LIN {X 0,Y 691.655,Z 288.187,A -85,B 0,C 180,E1 31271.101,E2 31271.101} C_VEL
LIN {X 0,Y 692.727,Z 290.872,A -85,B 0,C 180,E1 31270.983,E2 31270.983} C_VEL
LIN {X 0,Y 697.002,Z 308.209,A -85,B 0,C 180,E1 31270.448,E2 31270.448} C_VEL
LIN {X 0,Y 694.595,Z 554.038,A -85,B 0,C 180,E1 31267.412,E2 31267.412} C_VEL
LIN {X 0,Y 693.004,Z 720.794,A -85,B 0,C 180,E1 31265.381,E2 31265.381} C_VEL
LIN {X 0,Y 692.454,Z 746.763,A -85,B 0,C 180,E1 31264.93,E2 31264.93} C_VEL
LIN {X 0,Y 691.672,Z 770.938,A -85,B 0,C 180,E1 31264.354,E2 31264.354} C_VEL
LIN {X 0,Y 690.893,Z 792.668,A -85,B 0,C 180,E1 31263.712,E2 31263.712} C_VEL
LIN {X 0,Y 689.877,Z 818.249,A -85,B 0,C 180,E1 31262.792,E2 31262.792} C_VEL
LIN {X 0,Y 688.879,Z 840.235,A -85,B 0,C 180,E1 31261.844,E2 31261.844} C_VEL
LIN {X 0,Y 687.927,Z 859.99,A -85,B 0,C 180,E1 31260.869,E2 31260.869} C_VEL
LIN {X 0,Y 686.715,Z 883.646,A -85,B 0,C 180,E1 31259.529,E2 31259.529} C_VEL
LIN {X 0,Y 685.722,Z 903.008,A -85,B 0,C 180,E1 31258.269,E2 31258.269} C_VEL
LIN {X 0,Y 684.739,Z 922.512,A -85,B 0,C 180,E1 31256.847,E2 31256.847} C_VEL
LIN {X 0,Y 683.705,Z 942.533,A -85,B 0,C 180,E1 31255.187,E2 31255.187} C_VEL
LIN {X 0,Y 682.935,Z 959.025,A -85,B 0,C 180,E1 31253.651,E2 31253.651} C_VEL
LIN {X 0,Y 682.076,Z 977.766,A -85,B 0,C 180,E1 31251.68,E2 31251.68} C_VEL
LIN {X 0,Y 681.526,Z 991.915,A -85,B 0,C 180,E1 31249.989,E2 31249.989} C_VEL
LIN {X 0,Y 680.987,Z 1006.96,A -85,B 0,C 180,E1 31247.959,E2 31247.959} C_VEL
LIN {X 0,Y 680.597,Z 1019.263,A -85,B 0,C 180,E1 31246.033,E2 31246.033} C_VEL
LIN {X 0,Y 680.349,Z 1029.493,A -85,B 0,C 180,E1 31244.208,E2 31244.208} C_VEL
LIN {X 0,Y 680.126,Z 1040.171,A -85,B 0,C 180,E1 31241.964,E2 31241.964} C_VEL
LIN {X 0,Y 680.014,Z 1047.574,A -85,B 0,C 180,E1 31240.077,E2 31240.077} C_VEL
LIN {X 0,Y 679.956,Z 1053.149,A -85,B 0,C 180,E1 31238.371,E2 31238.371} C_VEL
LIN {X 0,Y 679.934,Z 1058.066,A -85,B 0,C 180,E1 31236.502,E2 31236.502} C_VEL
LIN {X 0,Y 679.908,Z 1062.337,A -85,B 0,C 180,E1 31234.217,E2 31234.217} C_VEL
LIN {X 0,Y 679.903,Z 1064.439,A -85,B 0,C 180,E1 31232.36,E2 31232.36} C_VEL
LIN {X 0,Y 679.893,Z 1065.35,A -85,B 0,C 180,E1 31230.59,E2 31230.59} C_VEL
LIN {X 0,Y 679.896,Z 1065.1,A -85,B 0,C 180,E1 31228.483,E2 31228.483} C_VEL
LIN {X 0,Y 679.907,Z 1063.128,A -85,B 0,C 180,E1 31226.374,E2 31226.374} C_VEL
LIN {X 0,Y 679.906,Z 1060.326,A -85,B 0,C 180,E1 31224.599,E2 31224.599} C_VEL
LIN {X 0,Y 679.946,Z 1056.414,A -85,B 0,C 180,E1 31222.82,E2 31222.82} C_VEL
LIN {X 0,Y 679.996,Z 1050.101,A -85,B 0,C 180,E1 31220.634,E2 31220.634} C_VEL
LIN {X 0,Y 680.095,Z 1042.663,A -85,B 0,C 180,E1 31218.638,E2 31218.638} C_VEL
LIN {X 0,Y 680.243,Z 1034.661,A -85,B 0,C 180,E1 31216.831,E2 31216.831} C_VEL
LIN {X 0,Y 680.475,Z 1023.917,A -85,B 0,C 180,E1 31214.751,E2 31214.751} C_VEL
LIN {X 0,Y 680.821,Z 1011.607,A -85,B 0,C 180,E1 31212.743,E2 31212.743} C_VEL
LIN {X 0,Y 681.259,Z 999.084,A -85,B 0,C 180,E1 31210.946,E2 31210.946} C_VEL
LIN {X 0,Y 681.869,Z 983.192,A -85,B 0,C 180,E1 31208.945,E2 31208.945} C_VEL
LIN {X 0,Y 682.513,Z 967.869,A -85,B 0,C 180,E1 31207.247,E2 31207.247} C_VEL
LIN {X 0,Y 683.4,Z 949.629,A -85,B 0,C 180,E1 31205.448,E2 31205.448} C_VEL
LIN {X 0,Y 684.27,Z 931.318,A -85,B 0,C 180,E1 31203.86,E2 31203.86} C_VEL
LIN {X 0,Y 685.293,Z 911.624,A -85,B 0,C 180,E1 31202.333,E2 31202.333} C_VEL
LIN {X 0,Y 686.389,Z 890.241,A -85,B 0,C 180,E1 31200.886,E2 31200.886} C_VEL
LIN {X 0,Y 687.364,Z 871.013,A -85,B 0,C 180,E1 31199.732,E2 31199.732} C_VEL
LIN {X 0,Y 688.556,Z 847.098,A -85,B 0,C 180,E1 31198.476,E2 31198.476} C_VEL
LIN {X 0,Y 689.557,Z 825.428,A -85,B 0,C 180,E1 31197.504,E2 31197.504} C_VEL
LIN {X 0,Y 690.438,Z 804.966,A -85,B 0,C 180,E1 31196.711,E2 31196.711} C_VEL
LIN {X 0,Y 691.403,Z 780.267,A -85,B 0,C 180,E1 31195.902,E2 31195.902} C_VEL
LIN {X 0,Y 692.129,Z 755.448,A -85,B 0,C 180,E1 31195.261,E2 31195.261} C_VEL
LIN {X 0,Y 692.718,Z 733.155,A -85,B 0,C 180,E1 31194.813,E2 31194.813} C_VEL
LIN {X 0,Y 693.254,Z 702.79,A -85,B 0,C 180,E1 31194.382,E2 31194.382} C_VEL
LIN {X 0,Y 695.461,Z 462.135,A -85,B 0,C 180,E1 31191.463,E2 31191.463} C_VEL
LIN {X 0,Y 696.866,Z 306.943,A -85,B 0,C 180,E1 31189.526,E2 31189.526} C_VEL
LIN {X 0,Y 691.957,Z 288.727,A -85,B 0,C 180,E1 31188.933,E2 31188.933} C_VEL
LIN {X 0,Y 690.695,Z 285.865,A -85,B 0,C 180,E1 31188.69,E2 31188.69} C_VEL
LIN {X 0,Y 681.985,Z 265.035,A -85,B 0,C 180,E1 31186.409,E2 31186.409} C_VEL
LIN {X 0,Y 680.481,Z 261.414,A -85,B 0,C 180,E1 31185.961,E2 31185.961} C_VEL
LIN {X 0,Y 680.519,Z 261.191,A -85,B 0,C 180,E1 31183.212,E2 31183.212} C_VEL
LIN {X 0,Y 680.458,Z 261.216,A -85,B 0,C 180,E1 31180.282,E2 31180.282} C_VEL
LIN {X 0,Y 680.458,Z 261.206,A -85,B 0,C 180,E1 31177.683,E2 31177.683} C_VEL
LIN {X 0,Y 680.502,Z 261.193,A -85,B 0,C 180,E1 31174.631,E2 31174.631} C_VEL
LIN {X 0,Y 680.449,Z 261.216,A -85,B 0,C 180,E1 31171.839,E2 31171.839} C_VEL
LIN {X 0,Y 680.517,Z 261.192,A -85,B 0,C 180,E1 31169.004,E2 31169.004} C_VEL
LIN {X 0,Y 680.459,Z 261.217,A -85,B 0,C 180,E1 31166.063,E2 31166.063} C_VEL
LIN {X 0,Y 680.458,Z 261.208,A -85,B 0,C 180,E1 31163.467,E2 31163.467} C_VEL
LIN {X 0,Y 680.512,Z 261.209,A -85,B 0,C 180,E1 31160.469,E2 31160.469} C_VEL
LIN {X 0,Y 680.45,Z 261.214,A -85,B 0,C 180,E1 31157.709,E2 31157.709} C_VEL
LIN {X 0,Y 680.488,Z 261.211,A -85,B 0,C 180,E1 31154.988,E2 31154.988} C_VEL
LIN {X 0,Y 680.467,Z 261.215,A -85,B 0,C 180,E1 31151.958,E2 31151.958} C_VEL
LIN {X 0,Y 680.454,Z 261.212,A -85,B 0,C 180,E1 31149.302,E2 31149.302} C_VEL
LIN {X 0,Y 680.524,Z 261.216,A -85,B 0,C 180,E1 31146.327,E2 31146.327} C_VEL
LIN {X 0,Y 680.449,Z 261.212,A -85,B 0,C 180,E1 31143.454,E2 31143.454} C_VEL
LIN {X 0,Y 680.498,Z 261.211,A -85,B 0,C 180,E1 31140.674,E2 31140.674} C_VEL
LIN {X 0,Y 680.46,Z 261.216,A -85,B 0,C 180,E1 31137.642,E2 31137.642} C_VEL
LIN {X 0,Y 680.455,Z 261.207,A -85,B 0,C 180,E1 31135.026,E2 31135.026} C_VEL
LIN {X 0,Y 680.514,Z 261.208,A -85,B 0,C 180,E1 31132.018,E2 31132.018} C_VEL
LIN {X 0,Y 680.449,Z 261.215,A -85,B 0,C 180,E1 31129.244,E2 31129.244} C_VEL
LIN {X 0,Y 680.48,Z 261.204,A -85,B 0,C 180,E1 31126.575,E2 31126.575} C_VEL
LIN {X 0,Y 680.468,Z 261.208,A -85,B 0,C 180,E1 31123.525,E2 31123.525} C_VEL
LIN {X 0,Y 680.451,Z 261.215,A -85,B 0,C 180,E1 31120.871,E2 31120.871} C_VEL
LIN {X 0,Y 680.53,Z 261.209,A -85,B 0,C 180,E1 31117.905,E2 31117.905} C_VEL
LIN {X 0,Y 680.447,Z 261.201,A -85,B 0,C 180,E1 31115.046,E2 31115.046} C_VEL
LIN {X 0,Y 680.479,Z 261.193,A -85,B 0,C 180,E1 31112.333,E2 31112.333} C_VEL
LIN {X 0,Y 680.498,Z 261.213,A -85,B 0,C 180,E1 31109.544,E2 31109.544} C_VEL
LIN {X 0,Y 679.438,Z 261.336,A -85,B 0,C 180,E1 31108.895,E2 31108.895} C_VEL
LIN {X 0,Y 673.022,Z 262.111,A -85,B 0,C 180,E1 31107.077,E2 31107.077} C_VEL
LIN {X 0,Y 672.51,Z 262.173,A -85,B 0,C 180,E1 31106.605,E2 31106.605} C_VEL
LIN {X 0,Y 672.581,Z 262.203,A -85,B 0,C 180,E1 31103.617,E2 31103.617} C_VEL
LIN {X 0,Y 672.511,Z 262.207,A -85,B 0,C 180,E1 31100.77,E2 31100.77} C_VEL
LIN {X 0,Y 672.551,Z 262.199,A -85,B 0,C 180,E1 31098.018,E2 31098.018} C_VEL
LIN {X 0,Y 672.519,Z 262.211,A -85,B 0,C 180,E1 31094.928,E2 31094.928} C_VEL
LIN {X 0,Y 672.516,Z 262.211,A -85,B 0,C 180,E1 31092.339,E2 31092.339} C_VEL
LIN {X 0,Y 672.546,Z 262.409,A -85,B 0,C 180,E1 31090.822,E2 31090.822} C_VEL
LIN {X 0,Y 675.389,Z 269.32,A -85,B 0,C 180,E1 31089.98,E2 31089.98} C_VEL
LIN {X 0,Y 679.147,Z 278.36,A -85,B 0,C 180,E1 31088.98,E2 31088.98} C_VEL
LIN {X 0,Y 689.647,Z 295.139,A -85,B 0,C 180,E1 31087.967,E2 31087.967} C_VEL
LIN {X 0,Y 690.879,Z 300.784,A -85,B 0,C 180,E1 31087.802,E2 31087.802} C_VEL
LIN {X 0,Y 688.209,Z 546.789,A -85,B 0,C 180,E1 31084.739,E2 31084.739} C_VEL
LIN {X 0,Y 686.469,Z 710.938,A -85,B 0,C 180,E1 31082.722,E2 31082.722} C_VEL
LIN {X 0,Y 685.844,Z 737.281,A -85,B 0,C 180,E1 31082.259,E2 31082.259} C_VEL
LIN {X 0,Y 685.014,Z 760.984,A -85,B 0,C 180,E1 31081.689,E2 31081.689} C_VEL
LIN {X 0,Y 684.18,Z 782.262,A -85,B 0,C 180,E1 31081.057,E2 31081.057} C_VEL
LIN {X 0,Y 683.101,Z 806.64,A -85,B 0,C 180,E1 31080.185,E2 31080.185} C_VEL
LIN {X 0,Y 681.937,Z 829.91,A -85,B 0,C 180,E1 31079.178,E2 31079.178} C_VEL
LIN {X 0,Y 680.867,Z 850.113,A -85,B 0,C 180,E1 31078.173,E2 31078.173} C_VEL
LIN {X 0,Y 679.511,Z 873.951,A -85,B 0,C 180,E1 31076.808,E2 31076.808} C_VEL
LIN {X 0,Y 678.374,Z 893.92,A -85,B 0,C 180,E1 31075.492,E2 31075.492} C_VEL
LIN {X 0,Y 677.213,Z 914.8,A -85,B 0,C 180,E1 31073.944,E2 31073.944} C_VEL
LIN {X 0,Y 676.092,Z 934.087,A -85,B 0,C 180,E1 31072.302,E2 31072.302} C_VEL
LIN {X 0,Y 675.237,Z 950.678,A -85,B 0,C 180,E1 31070.727,E2 31070.727} C_VEL
LIN {X 0,Y 674.302,Z 968.848,A -85,B 0,C 180,E1 31068.77,E2 31068.77} C_VEL
LIN {X 0,Y 673.674,Z 983.352,A -85,B 0,C 180,E1 31067.001,E2 31067.001} C_VEL
LIN {X 0,Y 673.066,Z 998.525,A -85,B 0,C 180,E1 31064.892,E2 31064.892} C_VEL
LIN {X 0,Y 672.666,Z 1009.999,A -85,B 0,C 180,E1 31063.058,E2 31063.058} C_VEL
LIN {X 0,Y 672.371,Z 1020.927,A -85,B 0,C 180,E1 31061.06,E2 31061.06} C_VEL
LIN {X 0,Y 672.144,Z 1030.836,A -85,B 0,C 180,E1 31058.9,E2 31058.9} C_VEL
LIN {X 0,Y 672.028,Z 1037.897,A -85,B 0,C 180,E1 31057.061,E2 31057.061} C_VEL
LIN {X 0,Y 671.964,Z 1043.795,A -85,B 0,C 180,E1 31055.208,E2 31055.208} C_VEL
LIN {X 0,Y 671.918,Z 1049.432,A -85,B 0,C 180,E1 31052.9,E2 31052.9} C_VEL
LIN {X 0,Y 671.919,Z 1052.713,A -85,B 0,C 180,E1 31050.938,E2 31050.938} C_VEL
LIN {X 0,Y 671.906,Z 1054.593,A -85,B 0,C 180,E1 31049.147,E2 31049.147} C_VEL
LIN {X 0,Y 671.908,Z 1055.491,A -85,B 0,C 180,E1 31047.014,E2 31047.014} C_VEL
LIN {X 0,Y 671.909,Z 1054.684,A -85,B 0,C 180,E1 31044.877,E2 31044.877} C_VEL
LIN {X 0,Y 671.917,Z 1052.852,A -85,B 0,C 180,E1 31043.077,E2 31043.077} C_VEL
LIN {X 0,Y 671.908,Z 1049.717,A -85,B 0,C 180,E1 31041.162,E2 31041.162} C_VEL
LIN {X 0,Y 671.96,Z 1044.22,A -85,B 0,C 180,E1 31038.846,E2 31038.846} C_VEL
LIN {X 0,Y 672.019,Z 1038.182,A -85,B 0,C 180,E1 31036.929,E2 31036.929} C_VEL
LIN {X 0,Y 672.14,Z 1031.512,A -85,B 0,C 180,E1 31035.175,E2 31035.175} C_VEL
LIN {X 0,Y 672.345,Z 1021.978,A -85,B 0,C 180,E1 31033.053,E2 31033.053} C_VEL
LIN {X 0,Y 672.658,Z 1010.349,A -85,B 0,C 180,E1 31030.912,E2 31030.912} C_VEL
LIN {X 0,Y 673.042,Z 999.136,A -85,B 0,C 180,E1 31029.112,E2 31029.112} C_VEL
LIN {X 0,Y 673.653,Z 983.784,A -85,B 0,C 180,E1 31026.964,E2 31026.964} C_VEL
LIN {X 0,Y 674.284,Z 969.258,A -85,B 0,C 180,E1 31025.187,E2 31025.187} C_VEL
LIN {X 0,Y 675.169,Z 952.248,A -85,B 0,C 180,E1 31023.338,E2 31023.338} C_VEL
LIN {X 0,Y 676.04,Z 935.141,A -85,B 0,C 180,E1 31021.704,E2 31021.704} C_VEL
LIN {X 0,Y 677.004,Z 917.895,A -85,B 0,C 180,E1 31020.221,E2 31020.221} C_VEL
LIN {X 0,Y 678.281,Z 895.722,A -85,B 0,C 180,E1 31018.544,E2 31018.544} C_VEL
LIN {X 0,Y 679.361,Z 876.399,A -85,B 0,C 180,E1 31017.256,E2 31017.256} C_VEL
LIN {X 0,Y 680.736,Z 852.619,A -85,B 0,C 180,E1 31015.869,E2 31015.869} C_VEL
LIN {X 0,Y 681.857,Z 831.556,A -85,B 0,C 180,E1 31014.809,E2 31014.809} C_VEL
LIN {X 0,Y 682.86,Z 811.527,A -85,B 0,C 180,E1 31013.928,E2 31013.928} C_VEL
LIN {X 0,Y 683.98,Z 787.389,A -85,B 0,C 180,E1 31013.019,E2 31013.019} C_VEL
LIN {X 0,Y 684.916,Z 763.254,A -85,B 0,C 180,E1 31012.282,E2 31012.282} C_VEL
LIN {X 0,Y 685.669,Z 741.656,A -85,B 0,C 180,E1 31011.748,E2 31011.748} C_VEL
LIN {X 0,Y 686.413,Z 715.552,A -85,B 0,C 180,E1 31011.254,E2 31011.254} C_VEL
LIN {X 0,Y 686.973,Z 669.627,A -85,B 0,C 180,E1 31010.667,E2 31010.667} C_VEL
LIN {X 0,Y 689.295,Z 440.854,A -85,B 0,C 180,E1 31007.861,E2 31007.861} C_VEL
LIN {X 0,Y 690.73,Z 299.325,A -85,B 0,C 180,E1 31006.077,E2 31006.077} C_VEL
LIN {X 0,Y 689.212,Z 294.353,A -85,B 0,C 180,E1 31005.901,E2 31005.901} C_VEL
LIN {X 0,Y 678.836,Z 277.664,A -85,B 0,C 180,E1 31004.874,E2 31004.874} C_VEL
LIN {X 0,Y 673.637,Z 265.405,A -85,B 0,C 180,E1 31003.462,E2 31003.462} C_VEL
LIN {X 0,Y 672.543,Z 262.387,A -85,B 0,C 180,E1 31003.08,E2 31003.08} C_VEL
LIN {X 0,Y 672.584,Z 262.19,A -85,B 0,C 180,E1 31000.17,E2 31000.17} C_VEL
LIN {X 0,Y 672.509,Z 262.194,A -85,B 0,C 180,E1 30997.303,E2 30997.303} C_VEL
LIN {X 0,Y 672.555,Z 262.193,A -85,B 0,C 180,E1 30994.55,E2 30994.55} C_VEL
LIN {X 0,Y 672.526,Z 262.2,A -85,B 0,C 180,E1 30991.557,E2 30991.557} C_VEL
LIN {X 0,Y 672.511,Z 262.204,A -85,B 0,C 180,E1 30988.993,E2 30988.993} C_VEL
LIN {X 0,Y 672.585,Z 262.176,A -85,B 0,C 180,E1 30986.107,E2 30986.107} C_VEL
LIN {X 0,Y 672.513,Z 262.204,A -85,B 0,C 180,E1 30983.204,E2 30983.204} C_VEL
LIN {X 0,Y 672.521,Z 262.188,A -85,B 0,C 180,E1 30980.632,E2 30980.632} C_VEL
LIN {X 0,Y 672.54,Z 262.203,A -85,B 0,C 180,E1 30977.477,E2 30977.477} C_VEL
LIN {X 0,Y 672.51,Z 262.195,A -85,B 0,C 180,E1 30974.817,E2 30974.817} C_VEL
LIN {X 0,Y 672.585,Z 262.19,A -85,B 0,C 180,E1 30971.926,E2 30971.926} C_VEL
LIN {X 0,Y 672.512,Z 262.198,A -85,B 0,C 180,E1 30968.981,E2 30968.981} C_VEL
LIN {X 0,Y 672.52,Z 262.174,A -85,B 0,C 180,E1 30966.402,E2 30966.402} C_VEL
LIN {X 0,Y 672.55,Z 262.2,A -85,B 0,C 180,E1 30963.324,E2 30963.324} C_VEL
LIN {X 0,Y 672.509,Z 262.185,A -85,B 0,C 180,E1 30960.596,E2 30960.596} C_VEL
LIN {X 0,Y 672.585,Z 262.196,A -85,B 0,C 180,E1 30957.7,E2 30957.7} C_VEL
LIN {X 0,Y 672.513,Z 262.195,A -85,B 0,C 180,E1 30954.711,E2 30954.711} C_VEL
LIN {X 0,Y 672.53,Z 262.178,A -85,B 0,C 180,E1 30952.052,E2 30952.052} C_VEL
LIN {X 0,Y 672.53,Z 262.199,A -85,B 0,C 180,E1 30948.889,E2 30948.889} C_VEL
LIN {X 0,Y 672.511,Z 262.177,A -85,B 0,C 180,E1 30946.238,E2 30946.238} C_VEL
LIN {X 0,Y 672.588,Z 262.201,A -85,B 0,C 180,E1 30943.326,E2 30943.326} C_VEL
LIN {X 0,Y 672.512,Z 262.186,A -85,B 0,C 180,E1 30940.456,E2 30940.456} C_VEL
LIN {X 0,Y 672.544,Z 262.196,A -85,B 0,C 180,E1 30937.721,E2 30937.721} C_VEL
LIN {X 0,Y 672.53,Z 262.199,A -85,B 0,C 180,E1 30934.647,E2 30934.647} C_VEL
LIN {X 0,Y 672.517,Z 262.203,A -85,B 0,C 180,E1 30931.977,E2 30931.977} C_VEL
LIN {X 0,Y 672.587,Z 262.19,A -85,B 0,C 180,E1 30929.044,E2 30929.044} C_VEL
LIN {X 0,Y 672.511,Z 262.191,A -85,B 0,C 180,E1 30926.113,E2 30926.113} C_VEL
LIN {X 0,Y 672.575,Z 262.186,A -85,B 0,C 180,E1 30923.255,E2 30923.255} C_VEL
LIN {X 0,Y 672.518,Z 262.206,A -85,B 0,C 180,E1 30920.234,E2 30920.234} C_VEL
LIN {X 0,Y 672.522,Z 262.208,A -85,B 0,C 180,E1 30917.64,E2 30917.64} C_VEL
LIN {X 0,Y 672.591,Z 262.407,A -85,B 0,C 180,E1 30914.594,E2 30914.594} C_VEL
LIN {X 0,Y 675.087,Z 268.808,A -85,B 0,C 180,E1 30913.837,E2 30913.837} C_VEL
LIN {X 0,Y 682.354,Z 285.802,A -85,B 0,C 180,E1 30911.928,E2 30911.928} C_VEL
LIN {X 0,Y 683.711,Z 288.641,A -85,B 0,C 180,E1 30911.673,E2 30911.673} C_VEL
LIN {X 0,Y 687.061,Z 294.502,A -85,B 0,C 180,E1 30911.345,E2 30911.345} C_VEL
LIN {X 0,Y 690.886,Z 310.252,A -85,B 0,C 180,E1 30910.854,E2 30910.854} C_VEL
LIN {X 0,Y 688.219,Z 556.025,A -85,B 0,C 180,E1 30907.794,E2 30907.794} C_VEL
LIN {X 0,Y 686.47,Z 720.881,A -85,B 0,C 180,E1 30905.768,E2 30905.768} C_VEL
LIN {X 0,Y 685.855,Z 747.02,A -85,B 0,C 180,E1 30905.31,E2 30905.31} C_VEL
LIN {X 0,Y 685.017,Z 770.919,A -85,B 0,C 180,E1 30904.735,E2 30904.735} C_VEL
LIN {X 0,Y 684.196,Z 791.933,A -85,B 0,C 180,E1 30904.112,E2 30904.112} C_VEL
LIN {X 0,Y 683.116,Z 816.377,A -85,B 0,C 180,E1 30903.241,E2 30903.241} C_VEL
LIN {X 0,Y 681.971,Z 839.227,A -85,B 0,C 180,E1 30902.255,E2 30902.255} C_VEL
LIN {X 0,Y 680.932,Z 858.899,A -85,B 0,C 180,E1 30901.282,E2 30901.282} C_VEL
LIN {X 0,Y 679.639,Z 882.174,A -85,B 0,C 180,E1 30899.965,E2 30899.965} C_VEL
LIN {X 0,Y 678.402,Z 903.283,A -85,B 0,C 180,E1 30898.582,E2 30898.582} C_VEL
LIN {X 0,Y 677.289,Z 923.369,A -85,B 0,C 180,E1 30897.099,E2 30897.099} C_VEL
LIN {X 0,Y 676.158,Z 942.892,A -85,B 0,C 180,E1 30895.455,E2 30895.455} C_VEL
LIN {X 0,Y 675.305,Z 959.023,A -85,B 0,C 180,E1 30893.935,E2 30893.935} C_VEL
LIN {X 0,Y 674.352,Z 977.768,A -85,B 0,C 180,E1 30891.941,E2 30891.941} C_VEL
LIN {X 0,Y 673.737,Z 991.914,A -85,B 0,C 180,E1 30890.23,E2 30890.23} C_VEL
LIN {X 0,Y 673.124,Z 1006.962,A -85,B 0,C 180,E1 30888.176,E2 30888.176} C_VEL
LIN {X 0,Y 672.684,Z 1019.35,A -85,B 0,C 180,E1 30886.213,E2 30886.213} C_VEL
LIN {X 0,Y 672.41,Z 1029.491,A -85,B 0,C 180,E1 30884.379,E2 30884.379} C_VEL
LIN {X 0,Y 672.157,Z 1040.172,A -85,B 0,C 180,E1 30882.108,E2 30882.108} C_VEL
LIN {X 0,Y 672.037,Z 1047.574,A -85,B 0,C 180,E1 30880.198,E2 30880.198} C_VEL
LIN {X 0,Y 671.961,Z 1053.405,A -85,B 0,C 180,E1 30878.385,E2 30878.385} C_VEL
LIN {X 0,Y 671.932,Z 1058.885,A -85,B 0,C 180,E1 30876.236,E2 30876.236} C_VEL
LIN {X 0,Y 671.913,Z 1062.564,A -85,B 0,C 180,E1 30874.096,E2 30874.096} C_VEL
LIN {X 0,Y 671.904,Z 1064.506,A -85,B 0,C 180,E1 30872.303,E2 30872.303} C_VEL
LIN {X 0,Y 671.892,Z 1065.395,A -85,B 0,C 180,E1 30870.426,E2 30870.426} C_VEL
LIN {X 0,Y 671.904,Z 1064.842,A -85,B 0,C 180,E1 30868.124,E2 30868.124} C_VEL
LIN {X 0,Y 671.911,Z 1063.015,A -85,B 0,C 180,E1 30866.246,E2 30866.246} C_VEL
LIN {X 0,Y 671.903,Z 1060.167,A -85,B 0,C 180,E1 30864.449,E2 30864.449} C_VEL
LIN {X 0,Y 671.949,Z 1056,A -85,B 0,C 180,E1 30862.562,E2 30862.562} C_VEL
LIN {X 0,Y 671.999,Z 1049.094,A -85,B 0,C 180,E1 30860.234,E2 30860.234} C_VEL
LIN {X 0,Y 672.131,Z 1042.308,A -85,B 0,C 180,E1 30858.415,E2 30858.415} C_VEL
LIN {X 0,Y 672.3,Z 1034.214,A -85,B 0,C 180,E1 30856.576,E2 30856.576} C_VEL
LIN {X 0,Y 672.597,Z 1022.886,A -85,B 0,C 180,E1 30854.391,E2 30854.391} C_VEL
LIN {X 0,Y 672.965,Z 1011.028,A -85,B 0,C 180,E1 30852.445,E2 30852.445} C_VEL
LIN {X 0,Y 673.481,Z 997.688,A -85,B 0,C 180,E1 30850.521,E2 30850.521} C_VEL
LIN {X 0,Y 674.192,Z 981.649,A -85,B 0,C 180,E1 30848.511,E2 30848.511} C_VEL
LIN {X 0,Y 674.879,Z 967.018,A -85,B 0,C 180,E1 30846.883,E2 30846.883} C_VEL
LIN {X 0,Y 675.928,Z 947.6,A -85,B 0,C 180,E1 30844.971,E2 30844.971} C_VEL
LIN {X 0,Y 676.829,Z 930.762,A -85,B 0,C 180,E1 30843.503,E2 30843.503} C_VEL
LIN {X 0,Y 678.02,Z 910.69,A -85,B 0,C 180,E1 30841.938,E2 30841.938} C_VEL
LIN {X 0,Y 679.23,Z 888.897,A -85,B 0,C 180,E1 30840.46,E2 30840.46} C_VEL
LIN {X 0,Y 680.369,Z 868.576,A -85,B 0,C 180,E1 30839.241,E2 30839.241} C_VEL
LIN {X 0,Y 681.735,Z 843.973,A -85,B 0,C 180,E1 30837.968,E2 30837.968} C_VEL
LIN {X 0,Y 682.775,Z 823.343,A -85,B 0,C 180,E1 30837.049,E2 30837.049} C_VEL
LIN {X 0,Y 683.767,Z 802.394,A -85,B 0,C 180,E1 30836.242,E2 30836.242} C_VEL
LIN {X 0,Y 684.827,Z 775.425,A -85,B 0,C 180,E1 30835.386,E2 30835.386} C_VEL
LIN {X 0,Y 685.596,Z 753.439,A -85,B 0,C 180,E1 30834.832,E2 30834.832} C_VEL
LIN {X 0,Y 686.302,Z 729.652,A -85,B 0,C 180,E1 30834.365,E2 30834.365} C_VEL
LIN {X 0,Y 686.824,Z 694.807,A -85,B 0,C 180,E1 30833.896,E2 30833.896} C_VEL
LIN {X 0,Y 689.235,Z 458.322,A -85,B 0,C 180,E1 30831,E2 30831} C_VEL
LIN {X 0,Y 690.749,Z 308.953,A -85,B 0,C 180,E1 30829.119,E2 30829.119} C_VEL
LIN {X 0,Y 686.523,Z 293.151,A -85,B 0,C 180,E1 30828.597,E2 30828.597} C_VEL
LIN {X 0,Y 683.09,Z 287.391,A -85,B 0,C 180,E1 30828.24,E2 30828.24} C_VEL
LIN {X 0,Y 675.482,Z 269.508,A -85,B 0,C 180,E1 30826.251,E2 30826.251} C_VEL
LIN {X 0,Y 672.607,Z 262.52,A -85,B 0,C 180,E1 30825.425,E2 30825.425} C_VEL
LIN {X 0,Y 672.54,Z 262.207,A -85,B 0,C 180,E1 30824.591,E2 30824.591} C_VEL
LIN {X 0,Y 672.515,Z 262.193,A -85,B 0,C 180,E1 30821.851,E2 30821.851} C_VEL
LIN {X 0,Y 672.584,Z 262.177,A -85,B 0,C 180,E1 30818.856,E2 30818.856} C_VEL
LIN {X 0,Y 672.513,Z 262.205,A -85,B 0,C 180,E1 30815.965,E2 30815.965} C_VEL
LIN {X 0,Y 672.564,Z 262.18,A -85,B 0,C 180,E1 30813.168,E2 30813.168} C_VEL
LIN {X 0,Y 672.521,Z 262.196,A -85,B 0,C 180,E1 30810.168,E2 30810.168} C_VEL
LIN {X 0,Y 672.518,Z 262.19,A -85,B 0,C 180,E1 30807.542,E2 30807.542} C_VEL
LIN {X 0,Y 672.57,Z 262.198,A -85,B 0,C 180,E1 30804.506,E2 30804.506} C_VEL
LIN {X 0,Y 672.512,Z 262.204,A -85,B 0,C 180,E1 30801.729,E2 30801.729} C_VEL
LIN {X 0,Y 672.568,Z 262.198,A -85,B 0,C 180,E1 30798.911,E2 30798.911} C_VEL
LIN {X 0,Y 672.517,Z 262.203,A -85,B 0,C 180,E1 30795.857,E2 30795.857} C_VEL
LIN {X 0,Y 672.522,Z 262.2,A -85,B 0,C 180,E1 30793.236,E2 30793.236} C_VEL
LIN {X 0,Y 672.547,Z 262.204,A -85,B 0,C 180,E1 30790.104,E2 30790.104} C_VEL
LIN {X 0,Y 672.51,Z 262.201,A -85,B 0,C 180,E1 30787.391,E2 30787.391} C_VEL
LIN {X 0,Y 672.585,Z 262.196,A -85,B 0,C 180,E1 30784.519,E2 30784.519} C_VEL
LIN {X 0,Y 672.513,Z 262.203,A -85,B 0,C 180,E1 30781.534,E2 30781.534} C_VEL
LIN {X 0,Y 672.529,Z 262.197,A -85,B 0,C 180,E1 30778.893,E2 30778.893} C_VEL
LIN {X 0,Y 672.531,Z 262.197,A -85,B 0,C 180,E1 30775.737,E2 30775.737} C_VEL
LIN {X 0,Y 672.512,Z 262.203,A -85,B 0,C 180,E1 30773.083,E2 30773.083} C_VEL
LIN {X 0,Y 672.588,Z 262.196,A -85,B 0,C 180,E1 30770.156,E2 30770.156} C_VEL
LIN {X 0,Y 672.51,Z 262.195,A -85,B 0,C 180,E1 30767.248,E2 30767.248} C_VEL
LIN {X 0,Y 672.53,Z 262.203,A -85,B 0,C 180,E1 30764.654,E2 30764.654} C_VEL
LIN {X 0,Y 672.527,Z 262.206,A -85,B 0,C 180,E1 30761.448,E2 30761.448} C_VEL
LIN {X 0,Y 672.515,Z 262.196,A -85,B 0,C 180,E1 30758.782,E2 30758.782} C_VEL
LIN {X 0,Y 672.577,Z 262.191,A -85,B 0,C 180,E1 30755.775,E2 30755.775} C_VEL
LIN {X 0,Y 672.507,Z 262.179,A -85,B 0,C 180,E1 30752.937,E2 30752.937} C_VEL
LIN {X 0,Y 672.552,Z 262.202,A -85,B 0,C 180,E1 30750.227,E2 30750.227} C_VEL
LIN {X 0,Y 672.516,Z 262.172,A -85,B 0,C 180,E1 30747.134,E2 30747.134} C_VEL
LIN {X 0,Y 672.51,Z 262.173,A -85,B 0,C 180,E1 30746.605,E2 30746.605} C_VEL
LIN {X 0,Y 671.56,Z 262.302,A -85,B 0,C 180,E1 30745.949,E2 30745.949} C_VEL
LIN {X 0,Y 665.112,Z 263.141,A -85,B 0,C 180,E1 30744.062,E2 30744.062} C_VEL
LIN {X 0,Y 664.643,Z 263.192,A -85,B 0,C 180,E1 30743.631,E2 30743.631} C_VEL
LIN {X 0,Y 664.572,Z 263.197,A -85,B 0,C 180,E1 30740.791,E2 30740.791} C_VEL
LIN {X 0,Y 664.605,Z 263.188,A -85,B 0,C 180,E1 30738.087,E2 30738.087} C_VEL
LIN {X 0,Y 664.586,Z 263.198,A -85,B 0,C 180,E1 30734.998,E2 30734.998} C_VEL
LIN {X 0,Y 664.575,Z 263.198,A -85,B 0,C 180,E1 30732.376,E2 30732.376} C_VEL
LIN {X 0,Y 664.685,Z 263.495,A -85,B 0,C 180,E1 30731.379,E2 30731.379} C_VEL
LIN {X 0,Y 670.815,Z 278.048,A -85,B 0,C 180,E1 30729.639,E2 30729.639} C_VEL
LIN {X 0,Y 684.181,Z 299.516,A -85,B 0,C 180,E1 30728.306,E2 30728.306} C_VEL
LIN {X 0,Y 684.794,Z 302.98,A -85,B 0,C 180,E1 30728.214,E2 30728.214} C_VEL
LIN {X 0,Y 681.873,Z 547.686,A -85,B 0,C 180,E1 30725.142,E2 30725.142} C_VEL
LIN {X 0,Y 679.968,Z 710.97,A -85,B 0,C 180,E1 30723.117,E2 30723.117} C_VEL
LIN {X 0,Y 679.28,Z 737.454,A -85,B 0,C 180,E1 30722.648,E2 30722.648} C_VEL
LIN {X 0,Y 678.393,Z 760.902,A -85,B 0,C 180,E1 30722.08,E2 30722.08} C_VEL
LIN {X 0,Y 677.559,Z 780.618,A -85,B 0,C 180,E1 30721.494,E2 30721.494} C_VEL
LIN {X 0,Y 676.486,Z 802.868,A -85,B 0,C 180,E1 30720.708,E2 30720.708} C_VEL
LIN {X 0,Y 675.119,Z 827.822,A -85,B 0,C 180,E1 30719.648,E2 30719.648} C_VEL
LIN {X 0,Y 673.935,Z 848.259,A -85,B 0,C 180,E1 30718.634,E2 30718.634} C_VEL
LIN {X 0,Y 672.584,Z 870.981,A -85,B 0,C 180,E1 30717.346,E2 30717.346} C_VEL
LIN {X 0,Y 671.148,Z 892.788,A -85,B 0,C 180,E1 30715.911,E2 30715.911} C_VEL
LIN {X 0,Y 669.994,Z 911.636,A -85,B 0,C 180,E1 30714.512,E2 30714.512} C_VEL
LIN {X 0,Y 668.709,Z 932.139,A -85,B 0,C 180,E1 30712.785,E2 30712.785} C_VEL
LIN {X 0,Y 667.726,Z 948.355,A -85,B 0,C 180,E1 30711.247,E2 30711.247} C_VEL
LIN {X 0,Y 666.762,Z 966.128,A -85,B 0,C 180,E1 30709.355,E2 30709.355} C_VEL
LIN {X 0,Y 665.988,Z 980.893,A -85,B 0,C 180,E1 30707.564,E2 30707.564} C_VEL
LIN {X 0,Y 665.367,Z 994.618,A -85,B 0,C 180,E1 30705.694,E2 30705.694} C_VEL
LIN {X 0,Y 664.827,Z 1008.169,A -85,B 0,C 180,E1 30703.569,E2 30703.569} C_VEL
LIN {X 0,Y 664.5,Z 1018.402,A -85,B 0,C 180,E1 30701.72,E2 30701.72} C_VEL
LIN {X 0,Y 664.231,Z 1028.467,A -85,B 0,C 180,E1 30699.619,E2 30699.619} C_VEL
LIN {X 0,Y 664.072,Z 1037.007,A -85,B 0,C 180,E1 30697.44,E2 30697.44} C_VEL
LIN {X 0,Y 663.966,Z 1042.891,A -85,B 0,C 180,E1 30695.617,E2 30695.617} C_VEL
LIN {X 0,Y 663.937,Z 1047.626,A -85,B 0,C 180,E1 30693.799,E2 30693.799} C_VEL
LIN {X 0,Y 663.897,Z 1051.969,A -85,B 0,C 180,E1 30691.553,E2 30691.553} C_VEL
LIN {X 0,Y 663.91,Z 1054.353,A -85,B 0,C 180,E1 30689.482,E2 30689.482} C_VEL
LIN {X 0,Y 663.896,Z 1055.322,A -85,B 0,C 180,E1 30687.669,E2 30687.669} C_VEL
LIN {X 0,Y 663.911,Z 1055.176,A -85,B 0,C 180,E1 30685.681,E2 30685.681} C_VEL
LIN {X 0,Y 663.907,Z 1053.371,A -85,B 0,C 180,E1 30683.427,E2 30683.427} C_VEL
LIN {X 0,Y 663.906,Z 1050.489,A -85,B 0,C 180,E1 30681.512,E2 30681.512} C_VEL
LIN {X 0,Y 663.949,Z 1046.802,A -85,B 0,C 180,E1 30679.764,E2 30679.764} C_VEL
LIN {X 0,Y 664.003,Z 1041.538,A -85,B 0,C 180,E1 30677.83,E2 30677.83} C_VEL
LIN {X 0,Y 664.139,Z 1033.33,A -85,B 0,C 180,E1 30675.482,E2 30675.482} C_VEL
LIN {X 0,Y 664.326,Z 1025.119,A -85,B 0,C 180,E1 30673.563,E2 30673.563} C_VEL
LIN {X 0,Y 664.586,Z 1015.231,A -85,B 0,C 180,E1 30671.582,E2 30671.582} C_VEL
LIN {X 0,Y 665.042,Z 1002.409,A -85,B 0,C 180,E1 30669.402,E2 30669.402} C_VEL
LIN {X 0,Y 665.563,Z 990.035,A -85,B 0,C 180,E1 30667.568,E2 30667.568} C_VEL
LIN {X 0,Y 666.337,Z 974.429,A -85,B 0,C 180,E1 30665.534,E2 30665.534} C_VEL
LIN {X 0,Y 667.122,Z 958.896,A -85,B 0,C 180,E1 30663.759,E2 30663.759} C_VEL
LIN {X 0,Y 668.19,Z 941.387,A -85,B 0,C 180,E1 30661.974,E2 30661.974} C_VEL
LIN {X 0,Y 669.303,Z 922.252,A -85,B 0,C 180,E1 30660.266,E2 30660.266} C_VEL
LIN {X 0,Y 670.438,Z 904.309,A -85,B 0,C 180,E1 30658.834,E2 30658.834} C_VEL
LIN {X 0,Y 671.894,Z 881.383,A -85,B 0,C 180,E1 30657.227,E2 30657.227} C_VEL
LIN {X 0,Y 673.073,Z 862.13,A -85,B 0,C 180,E1 30656.043,E2 30656.043} C_VEL
LIN {X 0,Y 674.532,Z 838.86,A -85,B 0,C 180,E1 30654.786,E2 30654.786} C_VEL
LIN {X 0,Y 675.825,Z 815.43,A -85,B 0,C 180,E1 30653.715,E2 30653.715} C_VEL
LIN {X 0,Y 676.85,Z 795.649,A -85,B 0,C 180,E1 30652.935,E2 30652.935} C_VEL
LIN {X 0,Y 677.876,Z 773.92,A -85,B 0,C 180,E1 30652.202,E2 30652.202} C_VEL
LIN {X 0,Y 678.875,Z 747.328,A -85,B 0,C 180,E1 30651.483,E2 30651.483} C_VEL
LIN {X 0,Y 679.574,Z 725.191,A -85,B 0,C 180,E1 30651.024,E2 30651.024} C_VEL
LIN {X 0,Y 680.197,Z 699.655,A -85,B 0,C 180,E1 30650.635,E2 30650.635} C_VEL
LIN {X 0,Y 682.922,Z 456.79,A -85,B 0,C 180,E1 30647.638,E2 30647.638} C_VEL
LIN {X 0,Y 684.655,Z 301.352,A -85,B 0,C 180,E1 30645.664,E2 30645.664} C_VEL
LIN {X 0,Y 683.59,Z 298.46,A -85,B 0,C 180,E1 30645.545,E2 30645.545} C_VEL
LIN {X 0,Y 670.7,Z 277.764,A -85,B 0,C 180,E1 30644.243,E2 30644.243} C_VEL
LIN {X 0,Y 664.682,Z 263.5,A -85,B 0,C 180,E1 30642.53,E2 30642.53} C_VEL
LIN {X 0,Y 664.571,Z 263.19,A -85,B 0,C 180,E1 30641.339,E2 30641.339} C_VEL
LIN {X 0,Y 664.63,Z 263.185,A -85,B 0,C 180,E1 30638.524,E2 30638.524} C_VEL
LIN {X 0,Y 664.58,Z 263.195,A -85,B 0,C 180,E1 30635.504,E2 30635.504} C_VEL
LIN {X 0,Y 664.579,Z 263.192,A -85,B 0,C 180,E1 30632.898,E2 30632.898} C_VEL
LIN {X 0,Y 664.625,Z 263.182,A -85,B 0,C 180,E1 30629.866,E2 30629.866} C_VEL
LIN {X 0,Y 664.572,Z 263.189,A -85,B 0,C 180,E1 30627.122,E2 30627.122} C_VEL
LIN {X 0,Y 664.635,Z 263.178,A -85,B 0,C 180,E1 30624.249,E2 30624.249} C_VEL
LIN {X 0,Y 664.578,Z 263.182,A -85,B 0,C 180,E1 30621.26,E2 30621.26} C_VEL
LIN {X 0,Y 664.585,Z 263.179,A -85,B 0,C 180,E1 30618.585,E2 30618.585} C_VEL
LIN {X 0,Y 664.601,Z 263.181,A -85,B 0,C 180,E1 30615.444,E2 30615.444} C_VEL
LIN {X 0,Y 664.57,Z 263.172,A -85,B 0,C 180,E1 30612.778,E2 30612.778} C_VEL
LIN {X 0,Y 664.65,Z 263.187,A -85,B 0,C 180,E1 30609.814,E2 30609.814} C_VEL
LIN {X 0,Y 664.569,Z 263.158,A -85,B 0,C 180,E1 30606.913,E2 30606.913} C_VEL
LIN {X 0,Y 664.597,Z 263.189,A -85,B 0,C 180,E1 30604.228,E2 30604.228} C_VEL
LIN {X 0,Y 664.584,Z 263.17,A -85,B 0,C 180,E1 30601.035,E2 30601.035} C_VEL
LIN {X 0,Y 664.578,Z 263.179,A -85,B 0,C 180,E1 30598.362,E2 30598.362} C_VEL
LIN {X 0,Y 664.631,Z 263.182,A -85,B 0,C 180,E1 30595.34,E2 30595.34} C_VEL
LIN {X 0,Y 664.568,Z 263.163,A -85,B 0,C 180,E1 30592.527,E2 30592.527} C_VEL
LIN {X 0,Y 664.636,Z 263.192,A -85,B 0,C 180,E1 30589.687,E2 30589.687} C_VEL
LIN {X 0,Y 664.577,Z 263.164,A -85,B 0,C 180,E1 30586.691,E2 30586.691} C_VEL
LIN {X 0,Y 664.587,Z 263.185,A -85,B 0,C 180,E1 30584.018,E2 30584.018} C_VEL
LIN {X 0,Y 664.599,Z 263.172,A -85,B 0,C 180,E1 30580.854,E2 30580.854} C_VEL
LIN {X 0,Y 664.574,Z 263.183,A -85,B 0,C 180,E1 30578.172,E2 30578.172} C_VEL
LIN {X 0,Y 664.651,Z 263.183,A -85,B 0,C 180,E1 30575.278,E2 30575.278} C_VEL
LIN {X 0,Y 664.575,Z 263.191,A -85,B 0,C 180,E1 30572.296,E2 30572.296} C_VEL
LIN {X 0,Y 664.604,Z 263.197,A -85,B 0,C 180,E1 30569.635,E2 30569.635} C_VEL
LIN {X 0,Y 664.584,Z 263.168,A -85,B 0,C 180,E1 30566.461,E2 30566.461} C_VEL
LIN {X 0,Y 664.579,Z 263.197,A -85,B 0,C 180,E1 30563.858,E2 30563.858} C_VEL
LIN {X 0,Y 664.636,Z 263.167,A -85,B 0,C 180,E1 30560.813,E2 30560.813} C_VEL
LIN {X 0,Y 664.574,Z 263.195,A -85,B 0,C 180,E1 30557.969,E2 30557.969} C_VEL
LIN {X 0,Y 664.663,Z 263.431,A -85,B 0,C 180,E1 30555.176,E2 30555.176} C_VEL
LIN {X 0,Y 673.862,Z 285.312,A -85,B 0,C 180,E1 30552.61,E2 30552.61} C_VEL
LIN {X 0,Y 675.209,Z 288.274,A -85,B 0,C 180,E1 30552.326,E2 30552.326} C_VEL
LIN {X 0,Y 681.574,Z 298.738,A -85,B 0,C 180,E1 30551.693,E2 30551.693} C_VEL
LIN {X 0,Y 684.804,Z 312.286,A -85,B 0,C 180,E1 30551.268,E2 30551.268} C_VEL
LIN {X 0,Y 681.881,Z 557.078,A -85,B 0,C 180,E1 30548.194,E2 30548.194} C_VEL
LIN {X 0,Y 679.969,Z 720.814,A -85,B 0,C 180,E1 30546.164,E2 30546.164} C_VEL
LIN {X 0,Y 679.293,Z 747.148,A -85,B 0,C 180,E1 30545.7,E2 30545.7} C_VEL
LIN {X 0,Y 678.402,Z 770.714,A -85,B 0,C 180,E1 30545.13,E2 30545.13} C_VEL
LIN {X 0,Y 677.532,Z 791.19,A -85,B 0,C 180,E1 30544.52,E2 30544.52} C_VEL
LIN {X 0,Y 676.433,Z 813.913,A -85,B 0,C 180,E1 30543.714,E2 30543.714} C_VEL
LIN {X 0,Y 675.098,Z 838.218,A -85,B 0,C 180,E1 30542.674,E2 30542.674} C_VEL
LIN {X 0,Y 673.94,Z 858.203,A -85,B 0,C 180,E1 30541.682,E2 30541.682} C_VEL
LIN {X 0,Y 672.605,Z 880.68,A -85,B 0,C 180,E1 30540.41,E2 30540.41} C_VEL
LIN {X 0,Y 671.209,Z 901.874,A -85,B 0,C 180,E1 30539.02,E2 30539.02} C_VEL
LIN {X 0,Y 670.057,Z 920.421,A -85,B 0,C 180,E1 30537.651,E2 30537.651} C_VEL
LIN {X 0,Y 668.75,Z 941.518,A -85,B 0,C 180,E1 30535.886,E2 30535.886} C_VEL
LIN {X 0,Y 667.738,Z 958.096,A -85,B 0,C 180,E1 30534.317,E2 30534.317} C_VEL
LIN {X 0,Y 666.809,Z 975.435,A -85,B 0,C 180,E1 30532.481,E2 30532.481} C_VEL
LIN {X 0,Y 665.974,Z 991.21,A -85,B 0,C 180,E1 30530.568,E2 30530.568} C_VEL
LIN {X 0,Y 665.346,Z 1005.108,A -85,B 0,C 180,E1 30528.669,E2 30528.669} C_VEL
LIN {X 0,Y 664.803,Z 1018.745,A -85,B 0,C 180,E1 30526.515,E2 30526.515} C_VEL
LIN {X 0,Y 664.485,Z 1029.031,A -85,B 0,C 180,E1 30524.643,E2 30524.643} C_VEL
LIN {X 0,Y 664.214,Z 1039.46,A -85,B 0,C 180,E1 30522.431,E2 30522.431} C_VEL
LIN {X 0,Y 664.067,Z 1047.27,A -85,B 0,C 180,E1 30520.41,E2 30520.41} C_VEL
LIN {X 0,Y 663.964,Z 1053.15,A -85,B 0,C 180,E1 30518.574,E2 30518.574} C_VEL
LIN {X 0,Y 663.936,Z 1058.066,A -85,B 0,C 180,E1 30516.659,E2 30516.659} C_VEL
LIN {X 0,Y 663.904,Z 1062.337,A -85,B 0,C 180,E1 30514.319,E2 30514.319} C_VEL
LIN {X 0,Y 663.905,Z 1064.439,A -85,B 0,C 180,E1 30512.417,E2 30512.417} C_VEL
LIN {X 0,Y 663.894,Z 1065.35,A -85,B 0,C 180,E1 30510.604,E2 30510.604} C_VEL
LIN {X 0,Y 663.895,Z 1065.099,A -85,B 0,C 180,E1 30508.447,E2 30508.447} C_VEL
LIN {X 0,Y 663.91,Z 1063.128,A -85,B 0,C 180,E1 30506.287,E2 30506.287} C_VEL
LIN {X 0,Y 663.905,Z 1060.326,A -85,B 0,C 180,E1 30504.469,E2 30504.469} C_VEL
LIN {X 0,Y 663.951,Z 1056.414,A -85,B 0,C 180,E1 30502.646,E2 30502.646} C_VEL
LIN {X 0,Y 664.009,Z 1050.306,A -85,B 0,C 180,E1 30500.466,E2 30500.466} C_VEL
LIN {X 0,Y 664.152,Z 1042.663,A -85,B 0,C 180,E1 30498.361,E2 30498.361} C_VEL
LIN {X 0,Y 664.337,Z 1034.537,A -85,B 0,C 180,E1 30496.482,E2 30496.482} C_VEL
LIN {X 0,Y 664.668,Z 1023.4,A -85,B 0,C 180,E1 30494.289,E2 30494.289} C_VEL
LIN {X 0,Y 665.075,Z 1011.607,A -85,B 0,C 180,E1 30492.321,E2 30492.321} C_VEL
LIN {X 0,Y 665.591,Z 999.366,A -85,B 0,C 180,E1 30490.519,E2 30490.519} C_VEL
LIN {X 0,Y 666.389,Z 983.188,A -85,B 0,C 180,E1 30488.432,E2 30488.432} C_VEL
LIN {X 0,Y 667.158,Z 968.308,A -85,B 0,C 180,E1 30486.741,E2 30486.741} C_VEL
LIN {X 0,Y 668.262,Z 950.135,A -85,B 0,C 180,E1 30484.901,E2 30484.901} C_VEL
LIN {X 0,Y 669.323,Z 931.87,A -85,B 0,C 180,E1 30483.278,E2 30483.278} C_VEL
LIN {X 0,Y 670.525,Z 913.13,A -85,B 0,C 180,E1 30481.79,E2 30481.79} C_VEL
LIN {X 0,Y 671.916,Z 890.973,A -85,B 0,C 180,E1 30480.246,E2 30480.246} C_VEL
LIN {X 0,Y 673.142,Z 870.925,A -85,B 0,C 180,E1 30479.018,E2 30479.018} C_VEL
LIN {X 0,Y 674.619,Z 847.224,A -85,B 0,C 180,E1 30477.753,E2 30477.753} C_VEL
LIN {X 0,Y 675.823,Z 825.421,A -85,B 0,C 180,E1 30476.759,E2 30476.759} C_VEL
LIN {X 0,Y 676.866,Z 805.349,A -85,B 0,C 180,E1 30475.969,E2 30475.969} C_VEL
LIN {X 0,Y 677.951,Z 782.316,A -85,B 0,C 180,E1 30475.196,E2 30475.196} C_VEL
LIN {X 0,Y 678.902,Z 756.539,A -85,B 0,C 180,E1 30474.51,E2 30474.51} C_VEL
LIN {X 0,Y 679.601,Z 734.474,A -85,B 0,C 180,E1 30474.056,E2 30474.056} C_VEL
LIN {X 0,Y 680.219,Z 707.836,A -85,B 0,C 180,E1 30473.657,E2 30473.657} C_VEL
LIN {X 0,Y 682.934,Z 465.741,A -85,B 0,C 180,E1 30470.669,E2 30470.669} C_VEL
LIN {X 0,Y 684.667,Z 310.936,A -85,B 0,C 180,E1 30468.704,E2 30468.704} C_VEL
LIN {X 0,Y 681.103,Z 297.645,A -85,B 0,C 180,E1 30468.257,E2 30468.257} C_VEL
LIN {X 0,Y 674.675,Z 287.31,A -85,B 0,C 180,E1 30467.599,E2 30467.599} C_VEL
LIN {X 0,Y 667.68,Z 270.691,A -85,B 0,C 180,E1 30465.712,E2 30465.712} C_VEL
LIN {X 0,Y 664.653,Z 263.381,A -85,B 0,C 180,E1 30464.808,E2 30464.808} C_VEL
LIN {X 0,Y 664.571,Z 263.176,A -85,B 0,C 180,E1 30462.031,E2 30462.031} C_VEL
LIN {X 0,Y 664.635,Z 263.168,A -85,B 0,C 180,E1 30459.187,E2 30459.187} C_VEL
LIN {X 0,Y 664.583,Z 263.196,A -85,B 0,C 180,E1 30456.248,E2 30456.248} C_VEL
LIN {X 0,Y 664.579,Z 263.169,A -85,B 0,C 180,E1 30453.62,E2 30453.62} C_VEL
LIN {X 0,Y 664.626,Z 263.186,A -85,B 0,C 180,E1 30450.564,E2 30450.564} C_VEL
LIN {X 0,Y 664.572,Z 263.179,A -85,B 0,C 180,E1 30447.788,E2 30447.788} C_VEL
LIN {X 0,Y 664.646,Z 263.192,A -85,B 0,C 180,E1 30444.886,E2 30444.886} C_VEL
LIN {X 0,Y 664.577,Z 263.194,A -85,B 0,C 180,E1 30441.909,E2 30441.909} C_VEL
LIN {X 0,Y 664.59,Z 263.188,A -85,B 0,C 180,E1 30439.238,E2 30439.238} C_VEL
LIN {X 0,Y 664.595,Z 263.191,A -85,B 0,C 180,E1 30436.071,E2 30436.071} C_VEL
LIN {X 0,Y 664.575,Z 263.19,A -85,B 0,C 180,E1 30433.397,E2 30433.397} C_VEL
LIN {X 0,Y 664.644,Z 263.194,A -85,B 0,C 180,E1 30430.401,E2 30430.401} C_VEL
LIN {X 0,Y 664.571,Z 263.191,A -85,B 0,C 180,E1 30427.521,E2 30427.521} C_VEL
LIN {X 0,Y 664.621,Z 263.188,A -85,B 0,C 180,E1 30424.746,E2 30424.746} C_VEL
LIN {X 0,Y 664.584,Z 263.193,A -85,B 0,C 180,E1 30421.724,E2 30421.724} C_VEL
LIN {X 0,Y 664.576,Z 263.187,A -85,B 0,C 180,E1 30419.138,E2 30419.138} C_VEL
LIN {X 0,Y 664.638,Z 263.184,A -85,B 0,C 180,E1 30416.118,E2 30416.118} C_VEL
LIN {X 0,Y 664.57,Z 263.193,A -85,B 0,C 180,E1 30413.26,E2 30413.26} C_VEL
LIN {X 0,Y 664.624,Z 263.181,A -85,B 0,C 180,E1 30410.474,E2 30410.474} C_VEL
LIN {X 0,Y 664.577,Z 263.184,A -85,B 0,C 180,E1 30407.399,E2 30407.399} C_VEL
LIN {X 0,Y 664.579,Z 263.193,A -85,B 0,C 180,E1 30404.824,E2 30404.824} C_VEL
LIN {X 0,Y 664.623,Z 263.193,A -85,B 0,C 180,E1 30401.764,E2 30401.764} C_VEL
LIN {X 0,Y 664.57,Z 263.185,A -85,B 0,C 180,E1 30399.017,E2 30399.017} C_VEL
LIN {X 0,Y 664.626,Z 263.191,A -85,B 0,C 180,E1 30396.222,E2 30396.222} C_VEL
LIN {X 0,Y 664.573,Z 263.162,A -85,B 0,C 180,E1 30393.151,E2 30393.151} C_VEL
LIN {X 0,Y 664.583,Z 263.192,A -85,B 0,C 180,E1 30390.529,E2 30390.529} C_VEL
LIN {X 0,Y 664.602,Z 263.158,A -85,B 0,C 180,E1 30387.406,E2 30387.406} C_VEL
LIN {X 0,Y 664.571,Z 263.193,A -85,B 0,C 180,E1 30384.707,E2 30384.707} C_VEL
LIN {X 0,Y 664.643,Z 263.192,A -85,B 0,C 180,E1 30383.631,E2 30383.631} C_VEL
LIN {X 0,Y 663.601,Z 263.311,A -85,B 0,C 180,E1 30382.967,E2 30382.967} C_VEL
LIN {X 0,Y 657.156,Z 264.123,A -85,B 0,C 180,E1 30381.106,E2 30381.106} C_VEL
LIN {X 0,Y 656.633,Z 264.186,A -85,B 0,C 180,E1 30380.621,E2 30380.621} C_VEL
LIN {X 0,Y 656.708,Z 264.177,A -85,B 0,C 180,E1 30377.702,E2 30377.702} C_VEL
LIN {X 0,Y 656.634,Z 264.189,A -85,B 0,C 180,E1 30374.709,E2 30374.709} C_VEL
LIN {X 0,Y 656.685,Z 264.357,A -85,B 0,C 180,E1 30372.025,E2 30372.025} C_VEL
LIN {X 0,Y 657.882,Z 267.446,A -85,B 0,C 180,E1 30371.602,E2 30371.602} C_VEL
LIN {X 0,Y 662.756,Z 278.624,A -85,B 0,C 180,E1 30370.269,E2 30370.269} C_VEL
LIN {X 0,Y 678.721,Z 303.778,A -85,B 0,C 180,E1 30368.655,E2 30368.655} C_VEL
LIN {X 0,Y 675.675,Z 540.217,A -85,B 0,C 180,E1 30365.656,E2 30365.656} C_VEL
LIN {X 0,Y 673.501,Z 710.899,A -85,B 0,C 180,E1 30363.521,E2 30363.521} C_VEL
LIN {X 0,Y 672.754,Z 737.44,A -85,B 0,C 180,E1 30363.048,E2 30363.048} C_VEL
LIN {X 0,Y 671.812,Z 760.64,A -85,B 0,C 180,E1 30362.483,E2 30362.483} C_VEL
LIN {X 0,Y 670.905,Z 780.415,A -85,B 0,C 180,E1 30361.893,E2 30361.893} C_VEL
LIN {X 0,Y 669.876,Z 800.216,A -85,B 0,C 180,E1 30361.195,E2 30361.195} C_VEL
LIN {X 0,Y 668.428,Z 825.004,A -85,B 0,C 180,E1 30360.16,E2 30360.16} C_VEL
LIN {X 0,Y 667.02,Z 846.874,A -85,B 0,C 180,E1 30359.079,E2 30359.079} C_VEL
LIN {X 0,Y 665.618,Z 868.552,A -85,B 0,C 180,E1 30357.851,E2 30357.851} C_VEL
LIN {X 0,Y 664.03,Z 891.193,A -85,B 0,C 180,E1 30356.369,E2 30356.369} C_VEL
LIN {X 0,Y 662.729,Z 909.797,A -85,B 0,C 180,E1 30354.989,E2 30354.989} C_VEL
LIN {X 0,Y 661.34,Z 930.591,A -85,B 0,C 180,E1 30353.241,E2 30353.241} C_VEL
LIN {X 0,Y 660.242,Z 946.939,A -85,B 0,C 180,E1 30351.686,E2 30351.686} C_VEL
LIN {X 0,Y 659.243,Z 963.282,A -85,B 0,C 180,E1 30349.954,E2 30349.954} C_VEL
LIN {X 0,Y 658.275,Z 979.808,A -85,B 0,C 180,E1 30347.96,E2 30347.96} C_VEL
LIN {X 0,Y 657.618,Z 993.014,A -85,B 0,C 180,E1 30346.155,E2 30346.155} C_VEL
LIN {X 0,Y 656.977,Z 1007.367,A -85,B 0,C 180,E1 30343.914,E2 30343.914} C_VEL
LIN {X 0,Y 656.579,Z 1017.687,A -85,B 0,C 180,E1 30342.042,E2 30342.042} C_VEL
LIN {X 0,Y 656.333,Z 1026.635,A -85,B 0,C 180,E1 30340.179,E2 30340.179} C_VEL
LIN {X 0,Y 656.096,Z 1036.01,A -85,B 0,C 180,E1 30337.86,E2 30337.86} C_VEL
LIN {X 0,Y 655.986,Z 1042.494,A -85,B 0,C 180,E1 30335.861,E2 30335.861} C_VEL
LIN {X 0,Y 655.945,Z 1047.303,A -85,B 0,C 180,E1 30334.021,E2 30334.021} C_VEL
LIN {X 0,Y 655.918,Z 1051.314,A -85,B 0,C 180,E1 30332.009,E2 30332.009} C_VEL
LIN {X 0,Y 655.917,Z 1054.246,A -85,B 0,C 180,E1 30329.651,E2 30329.651} C_VEL
LIN {X 0,Y 655.899,Z 1055.309,A -85,B 0,C 180,E1 30327.728,E2 30327.728} C_VEL
LIN {X 0,Y 655.915,Z 1055.211,A -85,B 0,C 180,E1 30325.804,E2 30325.804} C_VEL
LIN {X 0,Y 655.907,Z 1053.436,A -85,B 0,C 180,E1 30323.435,E2 30323.435} C_VEL
LIN {X 0,Y 655.907,Z 1050.581,A -85,B 0,C 180,E1 30321.496,E2 30321.496} C_VEL
LIN {X 0,Y 655.952,Z 1046.921,A -85,B 0,C 180,E1 30319.727,E2 30319.727} C_VEL
LIN {X 0,Y 656.005,Z 1041.943,A -85,B 0,C 180,E1 30317.858,E2 30317.858} C_VEL
LIN {X 0,Y 656.151,Z 1034.071,A -85,B 0,C 180,E1 30315.528,E2 30315.528} C_VEL
LIN {X 0,Y 656.356,Z 1025.768,A -85,B 0,C 180,E1 30313.54,E2 30313.54} C_VEL
LIN {X 0,Y 656.619,Z 1016.44,A -85,B 0,C 180,E1 30311.626,E2 30311.626} C_VEL
LIN {X 0,Y 657.131,Z 1003.49,A -85,B 0,C 180,E1 30309.356,E2 30309.356} C_VEL
LIN {X 0,Y 657.7,Z 991.059,A -85,B 0,C 180,E1 30307.474,E2 30307.474} C_VEL
LIN {X 0,Y 658.538,Z 975.814,A -85,B 0,C 180,E1 30305.436,E2 30305.436} C_VEL
LIN {X 0,Y 659.449,Z 959.376,A -85,B 0,C 180,E1 30303.527,E2 30303.527} C_VEL
LIN {X 0,Y 660.542,Z 942.87,A -85,B 0,C 180,E1 30301.817,E2 30301.817} C_VEL
LIN {X 0,Y 661.799,Z 923.451,A -85,B 0,C 180,E1 30300.044,E2 30300.044} C_VEL
LIN {X 0,Y 663.025,Z 905.681,A -85,B 0,C 180,E1 30298.603,E2 30298.603} C_VEL
LIN {X 0,Y 664.594,Z 883.341,A -85,B 0,C 180,E1 30297.001,E2 30297.001} C_VEL
LIN {X 0,Y 665.942,Z 863.063,A -85,B 0,C 180,E1 30295.733,E2 30295.733} C_VEL
LIN {X 0,Y 667.378,Z 841.776,A -85,B 0,C 180,E1 30294.562,E2 30294.562} C_VEL
LIN {X 0,Y 668.877,Z 817.79,A -85,B 0,C 180,E1 30293.432,E2 30293.432} C_VEL
LIN {X 0,Y 670.038,Z 797.147,A -85,B 0,C 180,E1 30292.601,E2 30292.601} C_VEL
LIN {X 0,Y 671.067,Z 777.176,A -85,B 0,C 180,E1 30291.913,E2 30291.913} C_VEL
LIN {X 0,Y 672.174,Z 752.873,A -85,B 0,C 180,E1 30291.216,E2 30291.216} C_VEL
LIN {X 0,Y 672.997,Z 727.585,A -85,B 0,C 180,E1 30290.666,E2 30290.666} C_VEL
LIN {X 0,Y 673.605,Z 705.295,A -85,B 0,C 180,E1 30290.309,E2 30290.309} C_VEL
LIN {X 0,Y 676.603,Z 467.206,A -85,B 0,C 180,E1 30287.339,E2 30287.339} C_VEL
LIN {X 0,Y 678.65,Z 303.667,A -85,B 0,C 180,E1 30285.248,E2 30285.248} C_VEL
LIN {X 0,Y 663.191,Z 279.282,A -85,B 0,C 180,E1 30283.687,E2 30283.687} C_VEL
LIN {X 0,Y 662.118,Z 277.41,A -85,B 0,C 180,E1 30283.522,E2 30283.522} C_VEL
LIN {X 0,Y 656.691,Z 264.38,A -85,B 0,C 180,E1 30281.894,E2 30281.894} C_VEL
LIN {X 0,Y 656.633,Z 264.188,A -85,B 0,C 180,E1 30279.307,E2 30279.307} C_VEL
LIN {X 0,Y 656.698,Z 264.174,A -85,B 0,C 180,E1 30276.428,E2 30276.428} C_VEL
LIN {X 0,Y 656.639,Z 264.179,A -85,B 0,C 180,E1 30273.441,E2 30273.441} C_VEL
LIN {X 0,Y 656.648,Z 264.171,A -85,B 0,C 180,E1 30270.773,E2 30270.773} C_VEL
LIN {X 0,Y 656.655,Z 264.176,A -85,B 0,C 180,E1 30267.575,E2 30267.575} C_VEL
LIN {X 0,Y 656.634,Z 264.163,A -85,B 0,C 180,E1 30264.852,E2 30264.852} C_VEL
LIN {X 0,Y 656.697,Z 264.168,A -85,B 0,C 180,E1 30261.809,E2 30261.809} C_VEL
LIN {X 0,Y 656.632,Z 264.165,A -85,B 0,C 180,E1 30258.926,E2 30258.926} C_VEL
LIN {X 0,Y 656.709,Z 264.173,A -85,B 0,C 180,E1 30255.997,E2 30255.997} C_VEL
LIN {X 0,Y 656.634,Z 264.158,A -85,B 0,C 180,E1 30253.025,E2 30253.025} C_VEL
LIN {X 0,Y 656.665,Z 264.184,A -85,B 0,C 180,E1 30250.262,E2 30250.262} C_VEL
LIN {X 0,Y 656.645,Z 264.143,A -85,B 0,C 180,E1 30247.173,E2 30247.173} C_VEL
LIN {X 0,Y 656.641,Z 264.177,A -85,B 0,C 180,E1 30244.454,E2 30244.454} C_VEL
LIN {X 0,Y 656.685,Z 264.157,A -85,B 0,C 180,E1 30241.396,E2 30241.396} C_VEL
LIN {X 0,Y 656.633,Z 264.167,A -85,B 0,C 180,E1 30238.604,E2 30238.604} C_VEL
LIN {X 0,Y 656.708,Z 264.174,A -85,B 0,C 180,E1 30235.634,E2 30235.634} C_VEL
LIN {X 0,Y 656.631,Z 264.148,A -85,B 0,C 180,E1 30232.651,E2 30232.651} C_VEL
LIN {X 0,Y 656.667,Z 264.179,A -85,B 0,C 180,E1 30229.915,E2 30229.915} C_VEL
LIN {X 0,Y 656.644,Z 264.151,A -85,B 0,C 180,E1 30226.796,E2 30226.796} C_VEL
LIN {X 0,Y 656.638,Z 264.172,A -85,B 0,C 180,E1 30224.183,E2 30224.183} C_VEL
LIN {X 0,Y 656.7,Z 264.159,A -85,B 0,C 180,E1 30221.168,E2 30221.168} C_VEL
LIN {X 0,Y 656.633,Z 264.171,A -85,B 0,C 180,E1 30218.26,E2 30218.26} C_VEL
LIN {X 0,Y 656.709,Z 264.172,A -85,B 0,C 180,E1 30215.343,E2 30215.343} C_VEL
LIN {X 0,Y 656.637,Z 264.18,A -85,B 0,C 180,E1 30212.326,E2 30212.326} C_VEL
LIN {X 0,Y 656.665,Z 264.186,A -85,B 0,C 180,E1 30209.633,E2 30209.633} C_VEL
LIN {X 0,Y 656.644,Z 264.154,A -85,B 0,C 180,E1 30206.444,E2 30206.444} C_VEL
LIN {X 0,Y 656.643,Z 264.185,A -85,B 0,C 180,E1 30203.785,E2 30203.785} C_VEL
LIN {X 0,Y 656.678,Z 264.16,A -85,B 0,C 180,E1 30200.669,E2 30200.669} C_VEL
LIN {X 0,Y 656.636,Z 264.184,A -85,B 0,C 180,E1 30197.932,E2 30197.932} C_VEL
LIN {X 0,Y 656.665,Z 264.387,A -85,B 0,C 180,E1 30195.804,E2 30195.804} C_VEL
LIN {X 0,Y 658.241,Z 268.072,A -85,B 0,C 180,E1 30195.306,E2 30195.306} C_VEL
LIN {X 0,Y 666.494,Z 287.492,A -85,B 0,C 180,E1 30193.031,E2 30193.031} C_VEL
LIN {X 0,Y 676.106,Z 302.921,A -85,B 0,C 180,E1 30192.047,E2 30192.047} C_VEL
LIN {X 0,Y 678.753,Z 314.232,A -85,B 0,C 180,E1 30191.689,E2 30191.689} C_VEL
LIN {X 0,Y 675.575,Z 558.492,A -85,B 0,C 180,E1 30188.597,E2 30188.597} C_VEL
LIN {X 0,Y 673.5,Z 720.831,A -85,B 0,C 180,E1 30186.568,E2 30186.568} C_VEL
LIN {X 0,Y 672.763,Z 747.276,A -85,B 0,C 180,E1 30186.097,E2 30186.097} C_VEL
LIN {X 0,Y 671.814,Z 770.602,A -85,B 0,C 180,E1 30185.529,E2 30185.529} C_VEL
LIN {X 0,Y 670.918,Z 790.14,A -85,B 0,C 180,E1 30184.947,E2 30184.947} C_VEL
LIN {X 0,Y 669.885,Z 810.091,A -85,B 0,C 180,E1 30184.244,E2 30184.244} C_VEL
LIN {X 0,Y 668.494,Z 834.094,A -85,B 0,C 180,E1 30183.248,E2 30183.248} C_VEL
LIN {X 0,Y 667.049,Z 856.398,A -85,B 0,C 180,E1 30182.15,E2 30182.15} C_VEL
LIN {X 0,Y 665.732,Z 876.674,A -85,B 0,C 180,E1 30181.008,E2 30181.008} C_VEL
LIN {X 0,Y 664.12,Z 900.07,A -85,B 0,C 180,E1 30179.493,E2 30179.493} C_VEL
LIN {X 0,Y 662.788,Z 918.892,A -85,B 0,C 180,E1 30178.105,E2 30178.105} C_VEL
LIN {X 0,Y 661.465,Z 938.982,A -85,B 0,C 180,E1 30176.434,E2 30176.434} C_VEL
LIN {X 0,Y 660.26,Z 956.705,A -85,B 0,C 180,E1 30174.754,E2 30174.754} C_VEL
LIN {X 0,Y 659.237,Z 973.483,A -85,B 0,C 180,E1 30172.976,E2 30172.976} C_VEL
LIN {X 0,Y 658.276,Z 989.795,A -85,B 0,C 180,E1 30171.006,E2 30171.006} C_VEL
LIN {X 0,Y 657.61,Z 1003.202,A -85,B 0,C 180,E1 30169.173,E2 30169.173} C_VEL
LIN {X 0,Y 656.984,Z 1017.184,A -85,B 0,C 180,E1 30166.99,E2 30166.99} C_VEL
LIN {X 0,Y 656.58,Z 1027.66,A -85,B 0,C 180,E1 30165.092,E2 30165.092} C_VEL
LIN {X 0,Y 656.328,Z 1036.698,A -85,B 0,C 180,E1 30163.21,E2 30163.21} C_VEL
LIN {X 0,Y 656.094,Z 1046.051,A -85,B 0,C 180,E1 30160.893,E2 30160.893} C_VEL
LIN {X 0,Y 655.988,Z 1052.385,A -85,B 0,C 180,E1 30158.944,E2 30158.944} C_VEL
LIN {X 0,Y 655.95,Z 1057.243,A -85,B 0,C 180,E1 30157.091,E2 30157.091} C_VEL
LIN {X 0,Y 655.92,Z 1061.282,A -85,B 0,C 180,E1 30155.072,E2 30155.072} C_VEL
LIN {X 0,Y 655.913,Z 1064.236,A -85,B 0,C 180,E1 30152.709,E2 30152.709} C_VEL
LIN {X 0,Y 655.9,Z 1065.305,A -85,B 0,C 180,E1 30150.786,E2 30150.786} C_VEL
LIN {X 0,Y 655.915,Z 1065.238,A -85,B 0,C 180,E1 30148.952,E2 30148.952} C_VEL
LIN {X 0,Y 655.907,Z 1063.692,A -85,B 0,C 180,E1 30146.679,E2 30146.679} C_VEL
LIN {X 0,Y 655.908,Z 1060.577,A -85,B 0,C 180,E1 30144.54,E2 30144.54} C_VEL
LIN {X 0,Y 655.954,Z 1056.827,A -85,B 0,C 180,E1 30142.732,E2 30142.732} C_VEL
LIN {X 0,Y 656.019,Z 1051.364,A -85,B 0,C 180,E1 30140.702,E2 30140.702} C_VEL
LIN {X 0,Y 656.166,Z 1043.369,A -85,B 0,C 180,E1 30138.396,E2 30138.396} C_VEL
LIN {X 0,Y 656.371,Z 1035.073,A -85,B 0,C 180,E1 30136.432,E2 30136.432} C_VEL
LIN {X 0,Y 656.698,Z 1024.867,A -85,B 0,C 180,E1 30134.366,E2 30134.366} C_VEL
LIN {X 0,Y 657.188,Z 1012.179,A -85,B 0,C 180,E1 30132.193,E2 30132.193} C_VEL
LIN {X 0,Y 657.749,Z 1000.011,A -85,B 0,C 180,E1 30130.369,E2 30130.369} C_VEL
LIN {X 0,Y 658.622,Z 983.956,A -85,B 0,C 180,E1 30128.258,E2 30128.258} C_VEL
LIN {X 0,Y 659.497,Z 968.721,A -85,B 0,C 180,E1 30126.5,E2 30126.5} C_VEL
LIN {X 0,Y 660.697,Z 950.641,A -85,B 0,C 180,E1 30124.641,E2 30124.641} C_VEL
LIN {X 0,Y 661.903,Z 931.869,A -85,B 0,C 180,E1 30122.955,E2 30122.955} C_VEL
LIN {X 0,Y 663.226,Z 913.128,A -85,B 0,C 180,E1 30121.451,E2 30121.451} C_VEL
LIN {X 0,Y 664.754,Z 890.658,A -85,B 0,C 180,E1 30119.87,E2 30119.87} C_VEL
LIN {X 0,Y 666.066,Z 871.199,A -85,B 0,C 180,E1 30118.669,E2 30118.669} C_VEL
LIN {X 0,Y 667.696,Z 847.228,A -85,B 0,C 180,E1 30117.377,E2 30117.377} C_VEL
LIN {X 0,Y 669.03,Z 824.873,A -85,B 0,C 180,E1 30116.353,E2 30116.353} C_VEL
LIN {X 0,Y 670.152,Z 804.956,A -85,B 0,C 180,E1 30115.565,E2 30115.565} C_VEL
LIN {X 0,Y 671.389,Z 780.385,A -85,B 0,C 180,E1 30114.741,E2 30114.741} C_VEL
LIN {X 0,Y 672.396,Z 755.625,A -85,B 0,C 180,E1 30114.091,E2 30114.091} C_VEL
LIN {X 0,Y 673.14,Z 733.872,A -85,B 0,C 180,E1 30113.644,E2 30113.644} C_VEL
LIN {X 0,Y 673.793,Z 706.201,A -85,B 0,C 180,E1 30113.232,E2 30113.232} C_VEL
LIN {X 0,Y 676.752,Z 464.85,A -85,B 0,C 180,E1 30110.227,E2 30110.227} C_VEL
LIN {X 0,Y 678.636,Z 312.98,A -85,B 0,C 180,E1 30108.284,E2 30108.284} C_VEL
LIN {X 0,Y 675.71,Z 302.091,A -85,B 0,C 180,E1 30107.911,E2 30107.911} C_VEL
LIN {X 0,Y 666.38,Z 287.23,A -85,B 0,C 180,E1 30106.944,E2 30106.944} C_VEL
LIN {X 0,Y 658.232,Z 268.061,A -85,B 0,C 180,E1 30104.691,E2 30104.691} C_VEL
LIN {X 0,Y 656.665,Z 264.382,A -85,B 0,C 180,E1 30104.204,E2 30104.204} C_VEL
LIN {X 0,Y 656.644,Z 264.168,A -85,B 0,C 180,E1 30101.716,E2 30101.716} C_VEL
LIN {X 0,Y 656.674,Z 264.154,A -85,B 0,C 180,E1 30098.63,E2 30098.63} C_VEL
LIN {X 0,Y 656.636,Z 264.184,A -85,B 0,C 180,E1 30095.892,E2 30095.892} C_VEL
LIN {X 0,Y 656.708,Z 264.156,A -85,B 0,C 180,E1 30092.927,E2 30092.927} C_VEL
LIN {X 0,Y 656.635,Z 264.172,A -85,B 0,C 180,E1 30089.953,E2 30089.953} C_VEL
LIN {X 0,Y 656.673,Z 264.165,A -85,B 0,C 180,E1 30087.181,E2 30087.181} C_VEL
LIN {X 0,Y 656.645,Z 264.176,A -85,B 0,C 180,E1 30084.085,E2 30084.085} C_VEL
LIN {X 0,Y 656.643,Z 264.181,A -85,B 0,C 180,E1 30081.436,E2 30081.436} C_VEL
LIN {X 0,Y 656.686,Z 264.183,A -85,B 0,C 180,E1 30078.372,E2 30078.372} C_VEL
LIN {X 0,Y 656.634,Z 264.18,A -85,B 0,C 180,E1 30075.546,E2 30075.546} C_VEL
LIN {X 0,Y 656.707,Z 264.171,A -85,B 0,C 180,E1 30072.665,E2 30072.665} C_VEL
LIN {X 0,Y 656.635,Z 264.18,A -85,B 0,C 180,E1 30069.643,E2 30069.643} C_VEL
LIN {X 0,Y 656.666,Z 264.177,A -85,B 0,C 180,E1 30066.89,E2 30066.89} C_VEL
LIN {X 0,Y 656.645,Z 264.179,A -85,B 0,C 180,E1 30063.754,E2 30063.754} C_VEL
LIN {X 0,Y 656.645,Z 264.179,A -85,B 0,C 180,E1 30061.047,E2 30061.047} C_VEL
LIN {X 0,Y 656.668,Z 264.184,A -85,B 0,C 180,E1 30057.906,E2 30057.906} C_VEL
LIN {X 0,Y 656.636,Z 264.173,A -85,B 0,C 180,E1 30055.108,E2 30055.108} C_VEL
LIN {X 0,Y 656.709,Z 264.173,A -85,B 0,C 180,E1 30052.124,E2 30052.124} C_VEL
LIN {X 0,Y 656.633,Z 264.183,A -85,B 0,C 180,E1 30049.205,E2 30049.205} C_VEL
LIN {X 0,Y 656.692,Z 264.169,A -85,B 0,C 180,E1 30046.349,E2 30046.349} C_VEL
LIN {X 0,Y 656.636,Z 264.172,A -85,B 0,C 180,E1 30043.295,E2 30043.295} C_VEL
LIN {X 0,Y 656.652,Z 264.181,A -85,B 0,C 180,E1 30040.613,E2 30040.613} C_VEL
LIN {X 0,Y 656.654,Z 264.184,A -85,B 0,C 180,E1 30037.435,E2 30037.435} C_VEL
LIN {X 0,Y 656.632,Z 264.163,A -85,B 0,C 180,E1 30034.757,E2 30034.757} C_VEL
LIN {X 0,Y 656.702,Z 264.16,A -85,B 0,C 180,E1 30031.736,E2 30031.736} C_VEL
LIN {X 0,Y 656.632,Z 264.176,A -85,B 0,C 180,E1 30028.921,E2 30028.921} C_VEL
LIN {X 0,Y 656.68,Z 264.145,A -85,B 0,C 180,E1 30026.082,E2 30026.082} C_VEL
LIN {X 0,Y 656.639,Z 264.178,A -85,B 0,C 180,E1 30023.024,E2 30023.024} C_VEL
LIN {X 0,Y 656.633,Z 264.186,A -85,B 0,C 180,E1 30020.621,E2 30020.621} C_VEL
LIN {X 0,Y 655.674,Z 264.308,A -85,B 0,C 180,E1 30019.95,E2 30019.95} C_VEL
LIN {X 0,Y 649.232,Z 265.104,A -85,B 0,C 180,E1 30018.016,E2 30018.016} C_VEL
LIN {X 0,Y 648.767,Z 265.169,A -85,B 0,C 180,E1 30017.575,E2 30017.575} C_VEL
LIN {X 0,Y 648.696,Z 265.178,A -85,B 0,C 180,E1 30014.592,E2 30014.592} C_VEL
LIN {X 0,Y 648.728,Z 265.424,A -85,B 0,C 180,E1 30012.618,E2 30012.618} C_VEL
LIN {X 0,Y 651.88,Z 272.681,A -85,B 0,C 180,E1 30011.669,E2 30011.669} C_VEL
LIN {X 0,Y 654.437,Z 278.783,A -85,B 0,C 180,E1 30010.958,E2 30010.958} C_VEL
LIN {X 0,Y 665.723,Z 296.06,A -85,B 0,C 180,E1 30009.773,E2 30009.773} C_VEL
LIN {X 0,Y 672.74,Z 307.507,A -85,B 0,C 180,E1 30009.059,E2 30009.059} C_VEL
LIN {X 0,Y 669.296,Z 550.096,A -85,B 0,C 180,E1 30005.961,E2 30005.961} C_VEL
LIN {X 0,Y 667.065,Z 711.035,A -85,B 0,C 180,E1 30003.93,E2 30003.93} C_VEL
LIN {X 0,Y 666.247,Z 737.786,A -85,B 0,C 180,E1 30003.449,E2 30003.449} C_VEL
LIN {X 0,Y 665.26,Z 760.503,A -85,B 0,C 180,E1 30002.892,E2 30002.892} C_VEL
LIN {X 0,Y 664.282,Z 780.213,A -85,B 0,C 180,E1 30002.3,E2 30002.3} C_VEL
LIN {X 0,Y 663.146,Z 800.491,A -85,B 0,C 180,E1 30001.58,E2 30001.58} C_VEL
LIN {X 0,Y 661.538,Z 825.799,A -85,B 0,C 180,E1 30000.51,E2 30000.51} C_VEL
LIN {X 0,Y 660.045,Z 847.155,A -85,B 0,C 180,E1 29999.444,E2 29999.444} C_VEL
LIN {X 0,Y 658.549,Z 868.459,A -85,B 0,C 180,E1 29998.226,E2 29998.226} C_VEL
LIN {X 0,Y 656.83,Z 891.211,A -85,B 0,C 180,E1 29996.722,E2 29996.722} C_VEL
LIN {X 0,Y 655.411,Z 909.728,A -85,B 0,C 180,E1 29995.336,E2 29995.336} C_VEL
LIN {X 0,Y 653.895,Z 930.532,A -85,B 0,C 180,E1 29993.57,E2 29993.57} C_VEL
LIN {X 0,Y 652.669,Z 947.339,A -85,B 0,C 180,E1 29991.95,E2 29991.95} C_VEL
LIN {X 0,Y 651.503,Z 964.797,A -85,B 0,C 180,E1 29990.071,E2 29990.071} C_VEL
LIN {X 0,Y 650.469,Z 980.813,A -85,B 0,C 180,E1 29988.09,E2 29988.09} C_VEL
LIN {X 0,Y 649.726,Z 994.538,A -85,B 0,C 180,E1 29986.173,E2 29986.173} C_VEL
LIN {X 0,Y 649.035,Z 1008.622,A -85,B 0,C 180,E1 29983.906,E2 29983.906} C_VEL
LIN {X 0,Y 648.618,Z 1018.796,A -85,B 0,C 180,E1 29982.012,E2 29982.012} C_VEL
LIN {X 0,Y 648.305,Z 1028.812,A -85,B 0,C 180,E1 29979.857,E2 29979.857} C_VEL
LIN {X 0,Y 648.097,Z 1037.269,A -85,B 0,C 180,E1 29977.624,E2 29977.624} C_VEL
LIN {X 0,Y 647.983,Z 1043.109,A -85,B 0,C 180,E1 29975.756,E2 29975.756} C_VEL
LIN {X 0,Y 647.942,Z 1048.007,A -85,B 0,C 180,E1 29973.805,E2 29973.805} C_VEL
LIN {X 0,Y 647.898,Z 1052.292,A -85,B 0,C 180,E1 29971.415,E2 29971.415} C_VEL
LIN {X 0,Y 647.91,Z 1054.411,A -85,B 0,C 180,E1 29969.469,E2 29969.469} C_VEL
LIN {X 0,Y 647.894,Z 1055.341,A -85,B 0,C 180,E1 29967.612,E2 29967.612} C_VEL
LIN {X 0,Y 647.899,Z 1055.133,A -85,B 0,C 180,E1 29965.486,E2 29965.486} C_VEL
LIN {X 0,Y 647.914,Z 1053.161,A -85,B 0,C 180,E1 29963.175,E2 29963.175} C_VEL
LIN {X 0,Y 647.907,Z 1050.353,A -85,B 0,C 180,E1 29961.301,E2 29961.301} C_VEL
LIN {X 0,Y 647.961,Z 1046.406,A -85,B 0,C 180,E1 29959.415,E2 29959.415} C_VEL
LIN {X 0,Y 648.029,Z 1040.236,A -85,B 0,C 180,E1 29957.162,E2 29957.162} C_VEL
LIN {X 0,Y 648.199,Z 1032.843,A -85,B 0,C 180,E1 29955.072,E2 29955.072} C_VEL
LIN {X 0,Y 648.426,Z 1024.76,A -85,B 0,C 180,E1 29953.148,E2 29953.148} C_VEL
LIN {X 0,Y 648.817,Z 1014.351,A -85,B 0,C 180,E1 29951.024,E2 29951.024} C_VEL
LIN {X 0,Y 649.346,Z 1001.893,A -85,B 0,C 180,E1 29948.88,E2 29948.88} C_VEL
LIN {X 0,Y 649.984,Z 989.462,A -85,B 0,C 180,E1 29947,E2 29947} C_VEL
LIN {X 0,Y 650.946,Z 972.943,A -85,B 0,C 180,E1 29944.819,E2 29944.819} C_VEL
LIN {X 0,Y 651.93,Z 958.129,A -85,B 0,C 180,E1 29943.099,E2 29943.099} C_VEL
LIN {X 0,Y 653.206,Z 940.043,A -85,B 0,C 180,E1 29941.227,E2 29941.227} C_VEL
LIN {X 0,Y 654.515,Z 921.812,A -85,B 0,C 180,E1 29939.574,E2 29939.574} C_VEL
LIN {X 0,Y 655.883,Z 903.895,A -85,B 0,C 180,E1 29938.119,E2 29938.119} C_VEL
LIN {X 0,Y 657.568,Z 881.191,A -85,B 0,C 180,E1 29936.498,E2 29936.498} C_VEL
LIN {X 0,Y 659.022,Z 861.495,A -85,B 0,C 180,E1 29935.269,E2 29935.269} C_VEL
LIN {X 0,Y 660.749,Z 838.11,A -85,B 0,C 180,E1 29933.992,E2 29933.992} C_VEL
LIN {X 0,Y 662.224,Z 815.087,A -85,B 0,C 180,E1 29932.925,E2 29932.925} C_VEL
LIN {X 0,Y 663.467,Z 794.676,A -85,B 0,C 180,E1 29932.111,E2 29932.111} C_VEL
LIN {X 0,Y 664.81,Z 769.805,A -85,B 0,C 180,E1 29931.276,E2 29931.276} C_VEL
LIN {X 0,Y 665.897,Z 745.498,A -85,B 0,C 180,E1 29930.637,E2 29930.637} C_VEL
LIN {X 0,Y 666.683,Z 723.969,A -85,B 0,C 180,E1 29930.192,E2 29930.192} C_VEL
LIN {X 0,Y 667.379,Z 696.546,A -85,B 0,C 180,E1 29929.779,E2 29929.779} C_VEL
LIN {X 0,Y 670.588,Z 455.801,A -85,B 0,C 180,E1 29926.755,E2 29926.755} C_VEL
LIN {X 0,Y 672.587,Z 307.065,A -85,B 0,C 180,E1 29924.833,E2 29924.833} C_VEL
LIN {X 0,Y 657.873,Z 283.832,A -85,B 0,C 180,E1 29923.318,E2 29923.318} C_VEL
LIN {X 0,Y 653.99,Z 277.883,A -85,B 0,C 180,E1 29922.872,E2 29922.872} C_VEL
LIN {X 0,Y 649.803,Z 268.338,A -85,B 0,C 180,E1 29921.663,E2 29921.663} C_VEL
LIN {X 0,Y 648.721,Z 265.358,A -85,B 0,C 180,E1 29921.248,E2 29921.248} C_VEL
LIN {X 0,Y 648.739,Z 265.165,A -85,B 0,C 180,E1 29918.609,E2 29918.609} C_VEL
LIN {X 0,Y 648.704,Z 265.173,A -85,B 0,C 180,E1 29915.528,E2 29915.528} C_VEL
LIN {X 0,Y 648.705,Z 265.17,A -85,B 0,C 180,E1 29912.856,E2 29912.856} C_VEL
LIN {X 0,Y 648.733,Z 265.16,A -85,B 0,C 180,E1 29909.756,E2 29909.756} C_VEL
LIN {X 0,Y 648.695,Z 265.162,A -85,B 0,C 180,E1 29907.011,E2 29907.011} C_VEL
LIN {X 0,Y 648.772,Z 265.158,A -85,B 0,C 180,E1 29904.009,E2 29904.009} C_VEL
LIN {X 0,Y 648.696,Z 265.159,A -85,B 0,C 180,E1 29901.142,E2 29901.142} C_VEL
LIN {X 0,Y 648.733,Z 265.155,A -85,B 0,C 180,E1 29898.326,E2 29898.326} C_VEL
LIN {X 0,Y 648.702,Z 265.159,A -85,B 0,C 180,E1 29895.191,E2 29895.191} C_VEL
LIN {X 0,Y 648.703,Z 265.148,A -85,B 0,C 180,E1 29892.553,E2 29892.553} C_VEL
LIN {X 0,Y 648.73,Z 265.163,A -85,B 0,C 180,E1 29889.403,E2 29889.403} C_VEL
LIN {X 0,Y 648.692,Z 265.132,A -85,B 0,C 180,E1 29886.639,E2 29886.639} C_VEL
LIN {X 0,Y 648.766,Z 265.168,A -85,B 0,C 180,E1 29883.623,E2 29883.623} C_VEL
LIN {X 0,Y 648.692,Z 265.144,A -85,B 0,C 180,E1 29880.707,E2 29880.707} C_VEL
LIN {X 0,Y 648.748,Z 265.157,A -85,B 0,C 180,E1 29877.88,E2 29877.88} C_VEL
LIN {X 0,Y 648.699,Z 265.161,A -85,B 0,C 180,E1 29874.782,E2 29874.782} C_VEL
LIN {X 0,Y 648.707,Z 265.138,A -85,B 0,C 180,E1 29872.115,E2 29872.115} C_VEL
LIN {X 0,Y 648.713,Z 265.165,A -85,B 0,C 180,E1 29868.891,E2 29868.891} C_VEL
LIN {X 0,Y 648.697,Z 265.135,A -85,B 0,C 180,E1 29866.177,E2 29866.177} C_VEL
LIN {X 0,Y 648.756,Z 265.167,A -85,B 0,C 180,E1 29863.157,E2 29863.157} C_VEL
LIN {X 0,Y 648.695,Z 265.145,A -85,B 0,C 180,E1 29860.271,E2 29860.271} C_VEL
LIN {X 0,Y 648.776,Z 265.167,A -85,B 0,C 180,E1 29857.242,E2 29857.242} C_VEL
LIN {X 0,Y 648.698,Z 265.167,A -85,B 0,C 180,E1 29854.334,E2 29854.334} C_VEL
LIN {X 0,Y 648.737,Z 265.163,A -85,B 0,C 180,E1 29851.559,E2 29851.559} C_VEL
LIN {X 0,Y 648.705,Z 265.155,A -85,B 0,C 180,E1 29848.47,E2 29848.47} C_VEL
LIN {X 0,Y 648.71,Z 265.156,A -85,B 0,C 180,E1 29845.706,E2 29845.706} C_VEL
LIN {X 0,Y 648.714,Z 265.136,A -85,B 0,C 180,E1 29842.495,E2 29842.495} C_VEL
LIN {X 0,Y 648.702,Z 265.176,A -85,B 0,C 180,E1 29839.772,E2 29839.772} C_VEL
LIN {X 0,Y 648.752,Z 265.163,A -85,B 0,C 180,E1 29836.674,E2 29836.674} C_VEL
LIN {X 0,Y 648.781,Z 265.57,A -85,B 0,C 180,E1 29836.401,E2 29836.401} C_VEL
LIN {X 0,Y 655.453,Z 281.083,A -85,B 0,C 180,E1 29834.443,E2 29834.443} C_VEL
LIN {X 0,Y 658.449,Z 287.72,A -85,B 0,C 180,E1 29833.679,E2 29833.679} C_VEL
LIN {X 0,Y 670.734,Z 307.38,A -85,B 0,C 180,E1 29832.398,E2 29832.398} C_VEL
LIN {X 0,Y 672.738,Z 316.323,A -85,B 0,C 180,E1 29832.117,E2 29832.117} C_VEL
LIN {X 0,Y 669.303,Z 559.843,A -85,B 0,C 180,E1 29829.009,E2 29829.009} C_VEL
LIN {X 0,Y 667.063,Z 721.025,A -85,B 0,C 180,E1 29826.976,E2 29826.976} C_VEL
LIN {X 0,Y 666.246,Z 747.796,A -85,B 0,C 180,E1 29826.493,E2 29826.493} C_VEL
LIN {X 0,Y 665.259,Z 770.535,A -85,B 0,C 180,E1 29825.936,E2 29825.936} C_VEL
LIN {X 0,Y 664.301,Z 789.852,A -85,B 0,C 180,E1 29825.356,E2 29825.356} C_VEL
LIN {X 0,Y 663.168,Z 810.088,A -85,B 0,C 180,E1 29824.64,E2 29824.64} C_VEL
LIN {X 0,Y 661.655,Z 834.303,A -85,B 0,C 180,E1 29823.626,E2 29823.626} C_VEL
LIN {X 0,Y 660.101,Z 856.394,A -85,B 0,C 180,E1 29822.53,E2 29822.53} C_VEL
LIN {X 0,Y 658.662,Z 876.677,A -85,B 0,C 180,E1 29821.379,E2 29821.379} C_VEL
LIN {X 0,Y 656.927,Z 900.067,A -85,B 0,C 180,E1 29819.849,E2 29819.849} C_VEL
LIN {X 0,Y 655.498,Z 918.602,A -85,B 0,C 180,E1 29818.469,E2 29818.469} C_VEL
LIN {X 0,Y 654.027,Z 938.886,A -85,B 0,C 180,E1 29816.768,E2 29816.768} C_VEL
LIN {X 0,Y 652.72,Z 956.704,A -85,B 0,C 180,E1 29815.06,E2 29815.06} C_VEL
LIN {X 0,Y 651.6,Z 972.944,A -85,B 0,C 180,E1 29813.322,E2 29813.322} C_VEL
LIN {X 0,Y 650.536,Z 989.796,A -85,B 0,C 180,E1 29811.268,E2 29811.268} C_VEL
LIN {X 0,Y 649.817,Z 1002.565,A -85,B 0,C 180,E1 29809.506,E2 29809.506} C_VEL
LIN {X 0,Y 649.15,Z 1016.143,A -85,B 0,C 180,E1 29807.387,E2 29807.387} C_VEL
LIN {X 0,Y 648.654,Z 1027.648,A -85,B 0,C 180,E1 29805.283,E2 29805.283} C_VEL
LIN {X 0,Y 648.377,Z 1036.697,A -85,B 0,C 180,E1 29803.375,E2 29803.375} C_VEL
LIN {X 0,Y 648.117,Z 1046.052,A -85,B 0,C 180,E1 29801.029,E2 29801.029} C_VEL
LIN {X 0,Y 647.995,Z 1052.64,A -85,B 0,C 180,E1 29798.966,E2 29798.966} C_VEL
LIN {X 0,Y 647.952,Z 1057.447,A -85,B 0,C 180,E1 29797.091,E2 29797.091} C_VEL
LIN {X 0,Y 647.909,Z 1061.757,A -85,B 0,C 180,E1 29794.869,E2 29794.869} C_VEL
LIN {X 0,Y 647.912,Z 1064.304,A -85,B 0,C 180,E1 29792.654,E2 29792.654} C_VEL
LIN {X 0,Y 647.9,Z 1065.305,A -85,B 0,C 180,E1 29790.796,E2 29790.796} C_VEL
LIN {X 0,Y 647.915,Z 1065.238,A -85,B 0,C 180,E1 29788.939,E2 29788.939} C_VEL
LIN {X 0,Y 647.906,Z 1063.693,A -85,B 0,C 180,E1 29786.638,E2 29786.638} C_VEL
LIN {X 0,Y 647.908,Z 1060.64,A -85,B 0,C 180,E1 29784.507,E2 29784.507} C_VEL
LIN {X 0,Y 647.956,Z 1057.034,A -85,B 0,C 180,E1 29782.731,E2 29782.731} C_VEL
LIN {X 0,Y 648.016,Z 1052.13,A -85,B 0,C 180,E1 29780.855,E2 29780.855} C_VEL
LIN {X 0,Y 648.169,Z 1044.428,A -85,B 0,C 180,E1 29778.522,E2 29778.522} C_VEL
LIN {X 0,Y 648.399,Z 1035.888,A -85,B 0,C 180,E1 29776.444,E2 29776.444} C_VEL
LIN {X 0,Y 648.694,Z 1026.724,A -85,B 0,C 180,E1 29774.535,E2 29774.535} C_VEL
LIN {X 0,Y 649.249,Z 1013.897,A -85,B 0,C 180,E1 29772.246,E2 29772.246} C_VEL
LIN {X 0,Y 649.878,Z 1001.296,A -85,B 0,C 180,E1 29770.309,E2 29770.309} C_VEL
LIN {X 0,Y 650.784,Z 986.251,A -85,B 0,C 180,E1 29768.267,E2 29768.267} C_VEL
LIN {X 0,Y 651.818,Z 969.564,A -85,B 0,C 180,E1 29766.303,E2 29766.303} C_VEL
LIN {X 0,Y 653.003,Z 952.99,A -85,B 0,C 180,E1 29764.564,E2 29764.564} C_VEL
LIN {X 0,Y 654.366,Z 933.787,A -85,B 0,C 180,E1 29762.788,E2 29762.788} C_VEL
LIN {X 0,Y 655.694,Z 916.168,A -85,B 0,C 180,E1 29761.341,E2 29761.341} C_VEL
LIN {X 0,Y 657.348,Z 894.582,A -85,B 0,C 180,E1 29759.767,E2 29759.767} C_VEL
LIN {X 0,Y 658.869,Z 873.432,A -85,B 0,C 180,E1 29758.428,E2 29758.428} C_VEL
LIN {X 0,Y 660.381,Z 852.796,A -85,B 0,C 180,E1 29757.28,E2 29757.28} C_VEL
LIN {X 0,Y 662.081,Z 827.674,A -85,B 0,C 180,E1 29756.081,E2 29756.081} C_VEL
LIN {X 0,Y 663.352,Z 806.765,A -85,B 0,C 180,E1 29755.235,E2 29755.235} C_VEL
LIN {X 0,Y 664.502,Z 786.009,A -85,B 0,C 180,E1 29754.518,E2 29754.518} C_VEL
LIN {X 0,Y 665.707,Z 760.034,A -85,B 0,C 180,E1 29753.786,E2 29753.786} C_VEL
LIN {X 0,Y 666.576,Z 736.583,A -85,B 0,C 180,E1 29753.284,E2 29753.284} C_VEL
LIN {X 0,Y 667.227,Z 713.667,A -85,B 0,C 180,E1 29752.919,E2 29752.919} C_VEL
LIN {X 0,Y 670.503,Z 472.473,A -85,B 0,C 180,E1 29749.886,E2 29749.886} C_VEL
LIN {X 0,Y 672.61,Z 314.952,A -85,B 0,C 180,E1 29747.854,E2 29747.854} C_VEL
LIN {X 0,Y 670.34,Z 306.576,A -85,B 0,C 180,E1 29747.56,E2 29747.56} C_VEL
LIN {X 0,Y 658.101,Z 287.123,A -85,B 0,C 180,E1 29746.267,E2 29746.267} C_VEL
LIN {X 0,Y 651.379,Z 271.906,A -85,B 0,C 180,E1 29744.425,E2 29744.425} C_VEL
LIN {X 0,Y 648.749,Z 265.377,A -85,B 0,C 180,E1 29743.592,E2 29743.592} C_VEL
LIN {X 0,Y 648.758,Z 265.171,A -85,B 0,C 180,E1 29740.805,E2 29740.805} C_VEL
LIN {X 0,Y 648.696,Z 265.152,A -85,B 0,C 180,E1 29737.953,E2 29737.953} C_VEL
LIN {X 0,Y 648.766,Z 265.145,A -85,B 0,C 180,E1 29734.983,E2 29734.983} C_VEL
LIN {X 0,Y 648.697,Z 265.174,A -85,B 0,C 180,E1 29732.022,E2 29732.022} C_VEL
LIN {X 0,Y 648.728,Z 265.144,A -85,B 0,C 180,E1 29729.248,E2 29729.248} C_VEL
LIN {X 0,Y 648.711,Z 265.174,A -85,B 0,C 180,E1 29726.157,E2 29726.157} C_VEL
LIN {X 0,Y 648.705,Z 265.163,A -85,B 0,C 180,E1 29723.433,E2 29723.433} C_VEL
LIN {X 0,Y 648.744,Z 265.162,A -85,B 0,C 180,E1 29720.385,E2 29720.385} C_VEL
LIN {X 0,Y 648.697,Z 265.169,A -85,B 0,C 180,E1 29717.585,E2 29717.585} C_VEL
LIN {X 0,Y 648.777,Z 265.169,A -85,B 0,C 180,E1 29714.549,E2 29714.549} C_VEL
LIN {X 0,Y 648.695,Z 265.169,A -85,B 0,C 180,E1 29711.559,E2 29711.559} C_VEL
LIN {X 0,Y 648.767,Z 265.159,A -85,B 0,C 180,E1 29708.598,E2 29708.598} C_VEL
LIN {X 0,Y 648.7,Z 265.169,A -85,B 0,C 180,E1 29705.661,E2 29705.661} C_VEL
LIN {X 0,Y 648.718,Z 265.165,A -85,B 0,C 180,E1 29702.916,E2 29702.916} C_VEL
LIN {X 0,Y 648.709,Z 265.164,A -85,B 0,C 180,E1 29699.735,E2 29699.735} C_VEL
LIN {X 0,Y 648.699,Z 265.17,A -85,B 0,C 180,E1 29697.084,E2 29697.084} C_VEL
LIN {X 0,Y 648.749,Z 265.171,A -85,B 0,C 180,E1 29693.984,E2 29693.984} C_VEL
LIN {X 0,Y 648.693,Z 265.161,A -85,B 0,C 180,E1 29691.222,E2 29691.222} C_VEL
LIN {X 0,Y 648.757,Z 265.169,A -85,B 0,C 180,E1 29688.352,E2 29688.352} C_VEL
LIN {X 0,Y 648.701,Z 265.173,A -85,B 0,C 180,E1 29685.358,E2 29685.358} C_VEL
LIN {X 0,Y 648.707,Z 265.158,A -85,B 0,C 180,E1 29682.693,E2 29682.693} C_VEL
LIN {X 0,Y 648.719,Z 265.162,A -85,B 0,C 180,E1 29679.52,E2 29679.52} C_VEL
LIN {X 0,Y 648.695,Z 265.171,A -85,B 0,C 180,E1 29676.855,E2 29676.855} C_VEL
LIN {X 0,Y 648.761,Z 265.124,A -85,B 0,C 180,E1 29673.845,E2 29673.845} C_VEL
LIN {X 0,Y 648.695,Z 265.172,A -85,B 0,C 180,E1 29670.922,E2 29670.922} C_VEL
LIN {X 0,Y 648.74,Z 265.144,A -85,B 0,C 180,E1 29668.129,E2 29668.129} C_VEL
LIN {X 0,Y 648.7,Z 265.166,A -85,B 0,C 180,E1 29665.013,E2 29665.013} C_VEL
LIN {X 0,Y 648.713,Z 265.16,A -85,B 0,C 180,E1 29662.272,E2 29662.272} C_VEL
LIN {X 0,Y 648.706,Z 265.161,A -85,B 0,C 180,E1 29659.048,E2 29659.048} C_VEL
LIN {X 0,Y 648.767,Z 265.169,A -85,B 0,C 180,E1 29657.575,E2 29657.575} C_VEL
LIN {X 0,Y 647.729,Z 265.31,A -85,B 0,C 180,E1 29656.895,E2 29656.895} C_VEL
LIN {X 0,Y 641.281,Z 266.109,A -85,B 0,C 180,E1 29654.988,E2 29654.988} C_VEL
LIN {X 0,Y 640.758,Z 266.167,A -85,B 0,C 180,E1 29654.491,E2 29654.491} C_VEL
LIN {X 0,Y 640.83,Z 266.376,A -85,B 0,C 180,E1 29653.26,E2 29653.26} C_VEL
LIN {X 0,Y 642.036,Z 269.61,A -85,B 0,C 180,E1 29652.817,E2 29652.817} C_VEL
LIN {X 0,Y 646.247,Z 278.902,A -85,B 0,C 180,E1 29651.66,E2 29651.66} C_VEL
LIN {X 0,Y 660.372,Z 300.45,A -85,B 0,C 180,E1 29650.142,E2 29650.142} C_VEL
LIN {X 0,Y 666.75,Z 310.954,A -85,B 0,C 180,E1 29649.478,E2 29649.478} C_VEL
LIN {X 0,Y 663.05,Z 552.129,A -85,B 0,C 180,E1 29646.372,E2 29646.372} C_VEL
LIN {X 0,Y 660.666,Z 711.067,A -85,B 0,C 180,E1 29644.349,E2 29644.349} C_VEL
LIN {X 0,Y 659.783,Z 737.931,A -85,B 0,C 180,E1 29643.861,E2 29643.861} C_VEL
LIN {X 0,Y 658.741,Z 760.367,A -85,B 0,C 180,E1 29643.308,E2 29643.308} C_VEL
LIN {X 0,Y 657.731,Z 779.291,A -85,B 0,C 180,E1 29642.739,E2 29642.739} C_VEL
LIN {X 0,Y 656.568,Z 798.62,A -85,B 0,C 180,E1 29642.055,E2 29642.055} C_VEL
LIN {X 0,Y 655.017,Z 822.514,A -85,B 0,C 180,E1 29641.061,E2 29641.061} C_VEL
LIN {X 0,Y 653.281,Z 845.281,A -85,B 0,C 180,E1 29639.931,E2 29639.931} C_VEL
LIN {X 0,Y 651.723,Z 865.216,A -85,B 0,C 180,E1 29638.799,E2 29638.799} C_VEL
LIN {X 0,Y 649.896,Z 888.372,A -85,B 0,C 180,E1 29637.289,E2 29637.289} C_VEL
LIN {X 0,Y 648.331,Z 907.272,A -85,B 0,C 180,E1 29635.878,E2 29635.878} C_VEL
LIN {X 0,Y 646.823,Z 925.815,A -85,B 0,C 180,E1 29634.328,E2 29634.328} C_VEL
LIN {X 0,Y 645.326,Z 945.014,A -85,B 0,C 180,E1 29632.501,E2 29632.501} C_VEL
LIN {X 0,Y 644.124,Z 960.693,A -85,B 0,C 180,E1 29630.823,E2 29630.823} C_VEL
LIN {X 0,Y 642.97,Z 977.638,A -85,B 0,C 180,E1 29628.778,E2 29628.778} C_VEL
LIN {X 0,Y 642.055,Z 991.685,A -85,B 0,C 180,E1 29626.838,E2 29626.838} C_VEL
LIN {X 0,Y 641.355,Z 1004.636,A -85,B 0,C 180,E1 29624.814,E2 29624.814} C_VEL
LIN {X 0,Y 640.788,Z 1016.715,A -85,B 0,C 180,E1 29622.618,E2 29622.618} C_VEL
LIN {X 0,Y 640.449,Z 1025.78,A -85,B 0,C 180,E1 29620.707,E2 29620.707} C_VEL
LIN {X 0,Y 640.206,Z 1034.253,A -85,B 0,C 180,E1 29618.623,E2 29618.623} C_VEL
LIN {X 0,Y 640.03,Z 1041.952,A -85,B 0,C 180,E1 29616.278,E2 29616.278} C_VEL
LIN {X 0,Y 639.959,Z 1046.863,A -85,B 0,C 180,E1 29614.391,E2 29614.391} C_VEL
LIN {X 0,Y 639.907,Z 1050.657,A -85,B 0,C 180,E1 29612.508,E2 29612.508} C_VEL
LIN {X 0,Y 639.908,Z 1053.806,A -85,B 0,C 180,E1 29610.269,E2 29610.269} C_VEL
LIN {X 0,Y 639.913,Z 1055.237,A -85,B 0,C 180,E1 29608.03,E2 29608.03} C_VEL
LIN {X 0,Y 639.9,Z 1055.305,A -85,B 0,C 180,E1 29606.147,E2 29606.147} C_VEL
LIN {X 0,Y 639.914,Z 1054.229,A -85,B 0,C 180,E1 29604.171,E2 29604.171} C_VEL
LIN {X 0,Y 639.923,Z 1051.406,A -85,B 0,C 180,E1 29601.825,E2 29601.825} C_VEL
LIN {X 0,Y 639.956,Z 1047.368,A -85,B 0,C 180,E1 29599.74,E2 29599.74} C_VEL
LIN {X 0,Y 640.018,Z 1042.495,A -85,B 0,C 180,E1 29597.824,E2 29597.824} C_VEL
LIN {X 0,Y 640.166,Z 1035.494,A -85,B 0,C 180,E1 29595.62,E2 29595.62} C_VEL
LIN {X 0,Y 640.429,Z 1026.641,A -85,B 0,C 180,E1 29593.398,E2 29593.398} C_VEL
LIN {X 0,Y 640.723,Z 1017.914,A -85,B 0,C 180,E1 29591.531,E2 29591.531} C_VEL
LIN {X 0,Y 641.246,Z 1006.78,A -85,B 0,C 180,E1 29589.461,E2 29589.461} C_VEL
LIN {X 0,Y 641.979,Z 993.076,A -85,B 0,C 180,E1 29587.278,E2 29587.278} C_VEL
LIN {X 0,Y 642.786,Z 980.111,A -85,B 0,C 180,E1 29585.46,E2 29585.46} C_VEL
LIN {X 0,Y 643.957,Z 962.927,A -85,B 0,C 180,E1 29583.337,E2 29583.337} C_VEL
LIN {X 0,Y 645.185,Z 946.778,A -85,B 0,C 180,E1 29581.59,E2 29581.59} C_VEL
LIN {X 0,Y 646.639,Z 928.433,A -85,B 0,C 180,E1 29579.812,E2 29579.812} C_VEL
LIN {X 0,Y 648.193,Z 908.889,A -85,B 0,C 180,E1 29578.159,E2 29578.159} C_VEL
LIN {X 0,Y 649.711,Z 890.57,A -85,B 0,C 180,E1 29576.779,E2 29576.779} C_VEL
LIN {X 0,Y 651.569,Z 867.425,A -85,B 0,C 180,E1 29575.243,E2 29575.243} C_VEL
LIN {X 0,Y 653.172,Z 846.631,A -85,B 0,C 180,E1 29574.051,E2 29574.051} C_VEL
LIN {X 0,Y 654.818,Z 824.84,A -85,B 0,C 180,E1 29572.959,E2 29572.959} C_VEL
LIN {X 0,Y 656.486,Z 800.143,A -85,B 0,C 180,E1 29571.914,E2 29571.914} C_VEL
LIN {X 0,Y 657.703,Z 779.878,A -85,B 0,C 180,E1 29571.191,E2 29571.191} C_VEL
LIN {X 0,Y 658.728,Z 760.603,A -85,B 0,C 180,E1 29570.609,E2 29570.609} C_VEL
LIN {X 0,Y 659.758,Z 738.401,A -85,B 0,C 180,E1 29570.06,E2 29570.06} C_VEL
LIN {X 0,Y 660.659,Z 711.283,A -85,B 0,C 180,E1 29569.564,E2 29569.564} C_VEL
LIN {X 0,Y 662.651,Z 579.341,A -85,B 0,C 180,E1 29567.883,E2 29567.883} C_VEL
LIN {X 0,Y 665.657,Z 375.174,A -85,B 0,C 180,E1 29565.262,E2 29565.262} C_VEL
LIN {X 0,Y 666.66,Z 310.472,A -85,B 0,C 180,E1 29564.418,E2 29564.418} C_VEL
LIN {X 0,Y 652.352,Z 288.078,A -85,B 0,C 180,E1 29562.916,E2 29562.916} C_VEL
LIN {X 0,Y 645.91,Z 278.111,A -85,B 0,C 180,E1 29562.177,E2 29562.177} C_VEL
LIN {X 0,Y 640.852,Z 266.481,A -85,B 0,C 180,E1 29560.621,E2 29560.621} C_VEL
LIN {X 0,Y 640.77,Z 266.153,A -85,B 0,C 180,E1 29559.709,E2 29559.709} C_VEL
LIN {X 0,Y 640.759,Z 266.147,A -85,B 0,C 180,E1 29557.038,E2 29557.038} C_VEL
LIN {X 0,Y 640.809,Z 266.141,A -85,B 0,C 180,E1 29553.96,E2 29553.96} C_VEL
LIN {X 0,Y 640.755,Z 266.151,A -85,B 0,C 180,E1 29551.099,E2 29551.099} C_VEL
LIN {X 0,Y 640.836,Z 266.155,A -85,B 0,C 180,E1 29548.113,E2 29548.113} C_VEL
LIN {X 0,Y 640.752,Z 266.135,A -85,B 0,C 180,E1 29545.116,E2 29545.116} C_VEL
LIN {X 0,Y 640.823,Z 266.152,A -85,B 0,C 180,E1 29542.185,E2 29542.185} C_VEL
LIN {X 0,Y 640.756,Z 266.138,A -85,B 0,C 180,E1 29539.129,E2 29539.129} C_VEL
LIN {X 0,Y 640.794,Z 266.162,A -85,B 0,C 180,E1 29536.312,E2 29536.312} C_VEL
LIN {X 0,Y 640.761,Z 266.128,A -85,B 0,C 180,E1 29533.162,E2 29533.162} C_VEL
LIN {X 0,Y 640.773,Z 266.161,A -85,B 0,C 180,E1 29530.429,E2 29530.429} C_VEL
LIN {X 0,Y 640.767,Z 266.116,A -85,B 0,C 180,E1 29527.171,E2 29527.171} C_VEL
LIN {X 0,Y 640.763,Z 266.154,A -85,B 0,C 180,E1 29524.475,E2 29524.475} C_VEL
LIN {X 0,Y 640.799,Z 266.132,A -85,B 0,C 180,E1 29521.341,E2 29521.341} C_VEL
LIN {X 0,Y 640.756,Z 266.142,A -85,B 0,C 180,E1 29518.569,E2 29518.569} C_VEL
LIN {X 0,Y 640.83,Z 266.148,A -85,B 0,C 180,E1 29515.525,E2 29515.525} C_VEL
LIN {X 0,Y 640.752,Z 266.122,A -85,B 0,C 180,E1 29512.558,E2 29512.558} C_VEL
LIN {X 0,Y 640.821,Z 266.158,A -85,B 0,C 180,E1 29509.663,E2 29509.663} C_VEL
LIN {X 0,Y 640.758,Z 266.124,A -85,B 0,C 180,E1 29506.647,E2 29506.647} C_VEL
LIN {X 0,Y 640.783,Z 266.15,A -85,B 0,C 180,E1 29503.874,E2 29503.874} C_VEL
LIN {X 0,Y 640.767,Z 266.135,A -85,B 0,C 180,E1 29500.682,E2 29500.682} C_VEL
LIN {X 0,Y 640.771,Z 266.149,A -85,B 0,C 180,E1 29497.91,E2 29497.91} C_VEL
LIN {X 0,Y 640.778,Z 266.153,A -85,B 0,C 180,E1 29494.687,E2 29494.687} C_VEL
LIN {X 0,Y 640.763,Z 266.157,A -85,B 0,C 180,E1 29491.985,E2 29491.985} C_VEL
LIN {X 0,Y 640.812,Z 266.142,A -85,B 0,C 180,E1 29488.904,E2 29488.904} C_VEL
LIN {X 0,Y 640.756,Z 266.136,A -85,B 0,C 180,E1 29486.037,E2 29486.037} C_VEL
LIN {X 0,Y 640.829,Z 266.127,A -85,B 0,C 180,E1 29483.023,E2 29483.023} C_VEL
LIN {X 0,Y 640.759,Z 266.157,A -85,B 0,C 180,E1 29480.107,E2 29480.107} C_VEL
LIN {X 0,Y 640.81,Z 266.201,A -85,B 0,C 180,E1 29477.253,E2 29477.253} C_VEL
LIN {X 0,Y 640.902,Z 266.637,A -85,B 0,C 180,E1 29477.054,E2 29477.054} C_VEL
LIN {X 0,Y 648.033,Z 283.152,A -85,B 0,C 180,E1 29474.909,E2 29474.909} C_VEL
LIN {X 0,Y 650.076,Z 287.73,A -85,B 0,C 180,E1 29474.386,E2 29474.386} C_VEL
LIN {X 0,Y 664.754,Z 310.63,A -85,B 0,C 180,E1 29472.822,E2 29472.822} C_VEL
LIN {X 0,Y 665.766,Z 313.378,A -85,B 0,C 180,E1 29472.702,E2 29472.702} C_VEL
LIN {X 0,Y 666.76,Z 318.407,A -85,B 0,C 180,E1 29472.552,E2 29472.552} C_VEL
LIN {X 0,Y 663.061,Z 561.427,A -85,B 0,C 180,E1 29469.425,E2 29469.425} C_VEL
LIN {X 0,Y 660.664,Z 720.964,A -85,B 0,C 180,E1 29467.396,E2 29467.396} C_VEL
LIN {X 0,Y 659.789,Z 747.794,A -85,B 0,C 180,E1 29466.909,E2 29466.909} C_VEL
LIN {X 0,Y 658.744,Z 770.315,A -85,B 0,C 180,E1 29466.354,E2 29466.354} C_VEL
LIN {X 0,Y 657.711,Z 789.701,A -85,B 0,C 180,E1 29465.77,E2 29465.77} C_VEL
LIN {X 0,Y 656.485,Z 810.085,A -85,B 0,C 180,E1 29465.044,E2 29465.044} C_VEL
LIN {X 0,Y 654.79,Z 835.191,A -85,B 0,C 180,E1 29463.979,E2 29463.979} C_VEL
LIN {X 0,Y 653.191,Z 856.39,A -85,B 0,C 180,E1 29462.917,E2 29462.917} C_VEL
LIN {X 0,Y 651.619,Z 876.679,A -85,B 0,C 180,E1 29461.757,E2 29461.757} C_VEL
LIN {X 0,Y 649.754,Z 900.065,A -85,B 0,C 180,E1 29460.213,E2 29460.213} C_VEL
LIN {X 0,Y 648.268,Z 917.992,A -85,B 0,C 180,E1 29458.866,E2 29458.866} C_VEL
LIN {X 0,Y 646.713,Z 937.401,A -85,B 0,C 180,E1 29457.235,E2 29457.235} C_VEL
LIN {X 0,Y 645.227,Z 956.239,A -85,B 0,C 180,E1 29455.42,E2 29455.42} C_VEL
LIN {X 0,Y 644.019,Z 972.097,A -85,B 0,C 180,E1 29453.711,E2 29453.711} C_VEL
LIN {X 0,Y 642.809,Z 989.812,A -85,B 0,C 180,E1 29451.535,E2 29451.535} C_VEL
LIN {X 0,Y 642.006,Z 1002.563,A -85,B 0,C 180,E1 29449.753,E2 29449.753} C_VEL
LIN {X 0,Y 641.28,Z 1016.145,A -85,B 0,C 180,E1 29447.607,E2 29447.607} C_VEL
LIN {X 0,Y 640.738,Z 1027.65,A -85,B 0,C 180,E1 29445.477,E2 29445.477} C_VEL
LIN {X 0,Y 640.425,Z 1036.696,A -85,B 0,C 180,E1 29443.544,E2 29443.544} C_VEL
LIN {X 0,Y 640.143,Z 1046.052,A -85,B 0,C 180,E1 29441.168,E2 29441.168} C_VEL
LIN {X 0,Y 640.013,Z 1052.641,A -85,B 0,C 180,E1 29439.079,E2 29439.079} C_VEL
LIN {X 0,Y 639.958,Z 1057.447,A -85,B 0,C 180,E1 29437.18,E2 29437.18} C_VEL
LIN {X 0,Y 639.913,Z 1061.757,A -85,B 0,C 180,E1 29434.93,E2 29434.93} C_VEL
LIN {X 0,Y 639.913,Z 1064.303,A -85,B 0,C 180,E1 29432.687,E2 29432.687} C_VEL
LIN {X 0,Y 639.901,Z 1065.305,A -85,B 0,C 180,E1 29430.806,E2 29430.806} C_VEL
LIN {X 0,Y 639.915,Z 1065.237,A -85,B 0,C 180,E1 29428.926,E2 29428.926} C_VEL
LIN {X 0,Y 639.907,Z 1063.693,A -85,B 0,C 180,E1 29426.596,E2 29426.596} C_VEL
LIN {X 0,Y 639.908,Z 1060.645,A -85,B 0,C 180,E1 29424.441,E2 29424.441} C_VEL
LIN {X 0,Y 639.96,Z 1057.034,A -85,B 0,C 180,E1 29422.639,E2 29422.639} C_VEL
LIN {X 0,Y 640.03,Z 1052.13,A -85,B 0,C 180,E1 29420.74,E2 29420.74} C_VEL
LIN {X 0,Y 640.201,Z 1044.427,A -85,B 0,C 180,E1 29418.377,E2 29418.377} C_VEL
LIN {X 0,Y 640.446,Z 1035.887,A -85,B 0,C 180,E1 29416.272,E2 29416.272} C_VEL
LIN {X 0,Y 640.794,Z 1026.61,A -85,B 0,C 180,E1 29414.316,E2 29414.316} C_VEL
LIN {X 0,Y 641.406,Z 1013.629,A -85,B 0,C 180,E1 29411.978,E2 29411.978} C_VEL
LIN {X 0,Y 642.081,Z 1001.294,A -85,B 0,C 180,E1 29410.06,E2 29410.06} C_VEL
LIN {X 0,Y 643.062,Z 986.252,A -85,B 0,C 180,E1 29407.993,E2 29407.993} C_VEL
LIN {X 0,Y 644.216,Z 969.562,A -85,B 0,C 180,E1 29406.006,E2 29406.006} C_VEL
LIN {X 0,Y 645.52,Z 952.526,A -85,B 0,C 180,E1 29404.198,E2 29404.198} C_VEL
LIN {X 0,Y 647.05,Z 932.976,A -85,B 0,C 180,E1 29402.381,E2 29402.381} C_VEL
LIN {X 0,Y 648.479,Z 915.557,A -85,B 0,C 180,E1 29400.942,E2 29400.942} C_VEL
LIN {X 0,Y 650.248,Z 893.889,A -85,B 0,C 180,E1 29399.353,E2 29399.353} C_VEL
LIN {X 0,Y 651.866,Z 873.428,A -85,B 0,C 180,E1 29398.049,E2 29398.049} C_VEL
LIN {X 0,Y 653.493,Z 852.792,A -85,B 0,C 180,E1 29396.891,E2 29396.891} C_VEL
LIN {X 0,Y 655.312,Z 827.671,A -85,B 0,C 180,E1 29395.682,E2 29395.682} C_VEL
LIN {X 0,Y 656.638,Z 807.472,A -85,B 0,C 180,E1 29394.857,E2 29394.857} C_VEL
LIN {X 0,Y 657.837,Z 787.411,A -85,B 0,C 180,E1 29394.155,E2 29394.155} C_VEL
LIN {X 0,Y 659.105,Z 763.375,A -85,B 0,C 180,E1 29393.453,E2 29393.453} C_VEL
LIN {X 0,Y 660.106,Z 737.719,A -85,B 0,C 180,E1 29392.887,E2 29392.887} C_VEL
LIN {X 0,Y 660.795,Z 715.488,A -85,B 0,C 180,E1 29392.526,E2 29392.526} C_VEL
LIN {X 0,Y 664.308,Z 477.108,A -85,B 0,C 180,E1 29389.5,E2 29389.5} C_VEL
LIN {X 0,Y 666.659,Z 317.029,A -85,B 0,C 180,E1 29387.42,E2 29387.42} C_VEL
LIN {X 0,Y 664.997,Z 311.038,A -85,B 0,C 180,E1 29387.203,E2 29387.203} C_VEL
LIN {X 0,Y 649.909,Z 287.467,A -85,B 0,C 180,E1 29385.598,E2 29385.598} C_VEL
LIN {X 0,Y 643.633,Z 273.253,A -85,B 0,C 180,E1 29383.858,E2 29383.858} C_VEL
LIN {X 0,Y 640.854,Z 266.354,A -85,B 0,C 180,E1 29382.952,E2 29382.952} C_VEL
LIN {X 0,Y 640.758,Z 266.153,A -85,B 0,C 180,E1 29380.01,E2 29380.01} C_VEL
LIN {X 0,Y 640.823,Z 266.147,A -85,B 0,C 180,E1 29377.125,E2 29377.125} C_VEL
LIN {X 0,Y 640.757,Z 266.128,A -85,B 0,C 180,E1 29374.044,E2 29374.044} C_VEL
LIN {X 0,Y 640.8,Z 266.16,A -85,B 0,C 180,E1 29371.201,E2 29371.201} C_VEL
LIN {X 0,Y 640.763,Z 266.132,A -85,B 0,C 180,E1 29368.116,E2 29368.116} C_VEL
LIN {X 0,Y 640.773,Z 266.161,A -85,B 0,C 180,E1 29365.379,E2 29365.379} C_VEL
LIN {X 0,Y 640.78,Z 266.162,A -85,B 0,C 180,E1 29362.187,E2 29362.187} C_VEL
LIN {X 0,Y 640.764,Z 266.156,A -85,B 0,C 180,E1 29359.413,E2 29359.413} C_VEL
LIN {X 0,Y 640.804,Z 266.15,A -85,B 0,C 180,E1 29356.312,E2 29356.312} C_VEL
LIN {X 0,Y 640.756,Z 266.157,A -85,B 0,C 180,E1 29353.537,E2 29353.537} C_VEL
LIN {X 0,Y 640.831,Z 266.158,A -85,B 0,C 180,E1 29350.519,E2 29350.519} C_VEL
LIN {X 0,Y 640.755,Z 266.157,A -85,B 0,C 180,E1 29347.532,E2 29347.532} C_VEL
LIN {X 0,Y 640.814,Z 266.15,A -85,B 0,C 180,E1 29344.654,E2 29344.654} C_VEL
LIN {X 0,Y 640.762,Z 266.16,A -85,B 0,C 180,E1 29341.61,E2 29341.61} C_VEL
LIN {X 0,Y 640.771,Z 266.152,A -85,B 0,C 180,E1 29338.927,E2 29338.927} C_VEL
LIN {X 0,Y 640.77,Z 266.15,A -85,B 0,C 180,E1 29335.652,E2 29335.652} C_VEL
LIN {X 0,Y 640.765,Z 266.159,A -85,B 0,C 180,E1 29332.919,E2 29332.919} C_VEL
LIN {X 0,Y 640.789,Z 266.163,A -85,B 0,C 180,E1 29329.753,E2 29329.753} C_VEL
LIN {X 0,Y 640.756,Z 266.147,A -85,B 0,C 180,E1 29327.014,E2 29327.014} C_VEL
LIN {X 0,Y 640.834,Z 266.152,A -85,B 0,C 180,E1 29324.061,E2 29324.061} C_VEL
LIN {X 0,Y 640.756,Z 266.161,A -85,B 0,C 180,E1 29321.06,E2 29321.06} C_VEL
LIN {X 0,Y 640.83,Z 266.148,A -85,B 0,C 180,E1 29318.104,E2 29318.104} C_VEL
LIN {X 0,Y 640.754,Z 266.14,A -85,B 0,C 180,E1 29315.081,E2 29315.081} C_VEL
LIN {X 0,Y 640.801,Z 266.128,A -85,B 0,C 180,E1 29312.189,E2 29312.189} C_VEL
LIN {X 0,Y 640.762,Z 266.154,A -85,B 0,C 180,E1 29309.11,E2 29309.11} C_VEL
LIN {X 0,Y 640.77,Z 266.117,A -85,B 0,C 180,E1 29306.361,E2 29306.361} C_VEL
LIN {X 0,Y 640.774,Z 266.156,A -85,B 0,C 180,E1 29303.178,E2 29303.178} C_VEL
LIN {X 0,Y 640.761,Z 266.164,A -85,B 0,C 180,E1 29300.456,E2 29300.456} C_VEL
LIN {X 0,Y 640.807,Z 266.162,A -85,B 0,C 180,E1 29297.375,E2 29297.375} C_VEL
LIN {X 0,Y 640.758,Z 266.167,A -85,B 0,C 180,E1 29294.491,E2 29294.491} C_VEL
LIN {X 0,Y 640.223,Z 266.835,A -85,B 0,C 180,E1 29294.095,E2 29294.095} C_VEL
LIN {X 0,Y 638.359,Z 269.589,A -85,B 0,C 180,E1 29293.555,E2 29293.555} C_VEL
LIN {X 0,Y 636.654,Z 273.951,A -85,B 0,C 180,E1 29292.996,E2 29292.996} C_VEL
LIN {X 0,Y 636.944,Z 277.132,A -85,B 0,C 180,E1 29292.608,E2 29292.608} C_VEL
LIN {X 0,Y 638.356,Z 279.592,A -85,B 0,C 180,E1 29292.343,E2 29292.343} C_VEL
LIN {X 0,Y 653.331,Z 302.247,A -85,B 0,C 180,E1 29290.699,E2 29290.699} C_VEL
LIN {X 0,Y 660.795,Z 314.365,A -85,B 0,C 180,E1 29289.904,E2 29289.904} C_VEL
LIN {X 0,Y 656.852,Z 553.578,A -85,B 0,C 180,E1 29286.798,E2 29286.798} C_VEL
LIN {X 0,Y 654.301,Z 711.099,A -85,B 0,C 180,E1 29284.776,E2 29284.776} C_VEL
LIN {X 0,Y 653.346,Z 738.17,A -85,B 0,C 180,E1 29284.28,E2 29284.28} C_VEL
LIN {X 0,Y 652.258,Z 760.231,A -85,B 0,C 180,E1 29283.732,E2 29283.732} C_VEL
LIN {X 0,Y 651.139,Z 779.809,A -85,B 0,C 180,E1 29283.139,E2 29283.139} C_VEL
LIN {X 0,Y 649.783,Z 800.951,A -85,B 0,C 180,E1 29282.378,E2 29282.378} C_VEL
LIN {X 0,Y 647.93,Z 826.315,A -85,B 0,C 180,E1 29281.284,E2 29281.284} C_VEL
LIN {X 0,Y 646.269,Z 846.923,A -85,B 0,C 180,E1 29280.239,E2 29280.239} C_VEL
LIN {X 0,Y 644.553,Z 867.49,A -85,B 0,C 180,E1 29279.049,E2 29279.049} C_VEL
LIN {X 0,Y 642.557,Z 890.56,A -85,B 0,C 180,E1 29277.503,E2 29277.503} C_VEL
LIN {X 0,Y 640.979,Z 908.391,A -85,B 0,C 180,E1 29276.147,E2 29276.147} C_VEL
LIN {X 0,Y 639.243,Z 928.366,A -85,B 0,C 180,E1 29274.445,E2 29274.445} C_VEL
LIN {X 0,Y 637.709,Z 946.322,A -85,B 0,C 180,E1 29272.688,E2 29272.688} C_VEL
LIN {X 0,Y 636.431,Z 961.888,A -85,B 0,C 180,E1 29270.99,E2 29270.99} C_VEL
LIN {X 0,Y 635.132,Z 979.342,A -85,B 0,C 180,E1 29268.828,E2 29268.828} C_VEL
LIN {X 0,Y 634.208,Z 992.584,A -85,B 0,C 180,E1 29266.958,E2 29266.958} C_VEL
LIN {X 0,Y 633.428,Z 1005.992,A -85,B 0,C 180,E1 29264.816,E2 29264.816} C_VEL
LIN {X 0,Y 632.848,Z 1017.375,A -85,B 0,C 180,E1 29262.686,E2 29262.686} C_VEL
LIN {X 0,Y 632.483,Z 1026.354,A -85,B 0,C 180,E1 29260.751,E2 29260.751} C_VEL
LIN {X 0,Y 632.203,Z 1035.415,A -85,B 0,C 180,E1 29258.458,E2 29258.458} C_VEL
LIN {X 0,Y 632.036,Z 1042.315,A -85,B 0,C 180,E1 29256.267,E2 29256.267} C_VEL
LIN {X 0,Y 631.962,Z 1047.156,A -85,B 0,C 180,E1 29254.355,E2 29254.355} C_VEL
LIN {X 0,Y 631.913,Z 1051.042,A -85,B 0,C 180,E1 29252.358,E2 29252.358} C_VEL
LIN {X 0,Y 631.928,Z 1054.128,A -85,B 0,C 180,E1 29249.909,E2 29249.909} C_VEL
LIN {X 0,Y 631.903,Z 1055.292,A -85,B 0,C 180,E1 29247.824,E2 29247.824} C_VEL
LIN {X 0,Y 631.911,Z 1055.25,A -85,B 0,C 180,E1 29245.917,E2 29245.917} C_VEL
LIN {X 0,Y 631.908,Z 1053.773,A -85,B 0,C 180,E1 29243.572,E2 29243.572} C_VEL
LIN {X 0,Y 631.908,Z 1050.697,A -85,B 0,C 180,E1 29241.354,E2 29241.354} C_VEL
LIN {X 0,Y 631.964,Z 1047.07,A -85,B 0,C 180,E1 29239.517,E2 29239.517} C_VEL
LIN {X 0,Y 632.037,Z 1042.127,A -85,B 0,C 180,E1 29237.576,E2 29237.576} C_VEL
LIN {X 0,Y 632.225,Z 1034.677,A -85,B 0,C 180,E1 29235.249,E2 29235.249} C_VEL
LIN {X 0,Y 632.492,Z 1026.051,A -85,B 0,C 180,E1 29233.089,E2 29233.089} C_VEL
LIN {X 0,Y 632.872,Z 1017.016,A -85,B 0,C 180,E1 29231.152,E2 29231.152} C_VEL
LIN {X 0,Y 633.521,Z 1004.294,A -85,B 0,C 180,E1 29228.812,E2 29228.812} C_VEL
LIN {X 0,Y 634.239,Z 992.143,A -85,B 0,C 180,E1 29226.887,E2 29226.887} C_VEL
LIN {X 0,Y 635.206,Z 978.348,A -85,B 0,C 180,E1 29224.948,E2 29224.948} C_VEL
LIN {X 0,Y 636.448,Z 961.68,A -85,B 0,C 180,E1 29222.896,E2 29222.896} C_VEL
LIN {X 0,Y 637.709,Z 946.312,A -85,B 0,C 180,E1 29221.221,E2 29221.221} C_VEL
LIN {X 0,Y 639.308,Z 927.615,A -85,B 0,C 180,E1 29219.397,E2 29219.397} C_VEL
LIN {X 0,Y 640.983,Z 908.337,A -85,B 0,C 180,E1 29217.758,E2 29217.758} C_VEL
LIN {X 0,Y 642.552,Z 890.649,A -85,B 0,C 180,E1 29216.413,E2 29216.413} C_VEL
LIN {X 0,Y 644.489,Z 868.354,A -85,B 0,C 180,E1 29214.914,E2 29214.914} C_VEL
LIN {X 0,Y 646.187,Z 847.91,A -85,B 0,C 180,E1 29213.725,E2 29213.725} C_VEL
LIN {X 0,Y 647.864,Z 827.036,A -85,B 0,C 180,E1 29212.66,E2 29212.66} C_VEL
LIN {X 0,Y 649.745,Z 801.641,A -85,B 0,C 180,E1 29211.559,E2 29211.559} C_VEL
LIN {X 0,Y 651.083,Z 780.847,A -85,B 0,C 180,E1 29210.806,E2 29210.806} C_VEL
LIN {X 0,Y 652.204,Z 761.222,A -85,B 0,C 180,E1 29210.206,E2 29210.206} C_VEL
LIN {X 0,Y 653.228,Z 740.576,A -85,B 0,C 180,E1 29209.686,E2 29209.686} C_VEL
LIN {X 0,Y 654.234,Z 714.739,A -85,B 0,C 180,E1 29209.189,E2 29209.189} C_VEL
LIN {X 0,Y 655.168,Z 662.99,A -85,B 0,C 180,E1 29208.506,E2 29208.506} C_VEL
LIN {X 0,Y 658.69,Z 437.209,A -85,B 0,C 180,E1 29205.608,E2 29205.608} C_VEL
LIN {X 0,Y 660.661,Z 313.849,A -85,B 0,C 180,E1 29203.987,E2 29203.987} C_VEL
LIN {X 0,Y 646.889,Z 292.278,A -85,B 0,C 180,E1 29202.506,E2 29202.506} C_VEL
LIN {X 0,Y 637.652,Z 278.424,A -85,B 0,C 180,E1 29201.432,E2 29201.432} C_VEL
LIN {X 0,Y 633.873,Z 270.081,A -85,B 0,C 180,E1 29200.297,E2 29200.297} C_VEL
LIN {X 0,Y 632.869,Z 267.295,A -85,B 0,C 180,E1 29199.869,E2 29199.869} C_VEL
LIN {X 0,Y 632.818,Z 267.134,A -85,B 0,C 180,E1 29197.127,E2 29197.127} C_VEL
LIN {X 0,Y 632.885,Z 267.126,A -85,B 0,C 180,E1 29194.116,E2 29194.116} C_VEL
LIN {X 0,Y 632.816,Z 267.141,A -85,B 0,C 180,E1 29191.216,E2 29191.216} C_VEL
LIN {X 0,Y 632.883,Z 267.149,A -85,B 0,C 180,E1 29188.292,E2 29188.292} C_VEL
LIN {X 0,Y 632.816,Z 267.119,A -85,B 0,C 180,E1 29185.253,E2 29185.253} C_VEL
LIN {X 0,Y 632.851,Z 267.151,A -85,B 0,C 180,E1 29182.44,E2 29182.44} C_VEL
LIN {X 0,Y 632.825,Z 267.12,A -85,B 0,C 180,E1 29179.283,E2 29179.283} C_VEL
LIN {X 0,Y 632.834,Z 267.152,A -85,B 0,C 180,E1 29176.523,E2 29176.523} C_VEL
LIN {X 0,Y 632.827,Z 267.113,A -85,B 0,C 180,E1 29173.244,E2 29173.244} C_VEL
LIN {X 0,Y 632.83,Z 267.15,A -85,B 0,C 180,E1 29170.469,E2 29170.469} C_VEL
LIN {X 0,Y 632.837,Z 267.102,A -85,B 0,C 180,E1 29167.262,E2 29167.262} C_VEL
LIN {X 0,Y 632.826,Z 267.143,A -85,B 0,C 180,E1 29164.44,E2 29164.44} C_VEL
LIN {X 0,Y 632.85,Z 267.12,A -85,B 0,C 180,E1 29161.267,E2 29161.267} C_VEL
LIN {X 0,Y 632.82,Z 267.131,A -85,B 0,C 180,E1 29158.461,E2 29158.461} C_VEL
LIN {X 0,Y 632.878,Z 267.136,A -85,B 0,C 180,E1 29155.378,E2 29155.378} C_VEL
LIN {X 0,Y 632.814,Z 267.109,A -85,B 0,C 180,E1 29152.464,E2 29152.464} C_VEL
LIN {X 0,Y 632.891,Z 267.143,A -85,B 0,C 180,E1 29149.44,E2 29149.44} C_VEL
LIN {X 0,Y 632.814,Z 267.109,A -85,B 0,C 180,E1 29146.476,E2 29146.476} C_VEL
LIN {X 0,Y 632.885,Z 267.14,A -85,B 0,C 180,E1 29143.534,E2 29143.534} C_VEL
LIN {X 0,Y 632.821,Z 267.12,A -85,B 0,C 180,E1 29140.525,E2 29140.525} C_VEL
LIN {X 0,Y 632.851,Z 267.138,A -85,B 0,C 180,E1 29137.716,E2 29137.716} C_VEL
LIN {X 0,Y 632.829,Z 267.143,A -85,B 0,C 180,E1 29134.547,E2 29134.547} C_VEL
LIN {X 0,Y 632.834,Z 267.143,A -85,B 0,C 180,E1 29131.808,E2 29131.808} C_VEL
LIN {X 0,Y 632.834,Z 267.129,A -85,B 0,C 180,E1 29128.562,E2 29128.562} C_VEL
LIN {X 0,Y 632.828,Z 267.128,A -85,B 0,C 180,E1 29125.771,E2 29125.771} C_VEL
LIN {X 0,Y 632.85,Z 267.109,A -85,B 0,C 180,E1 29122.629,E2 29122.629} C_VEL
LIN {X 0,Y 632.822,Z 267.153,A -85,B 0,C 180,E1 29119.86,E2 29119.86} C_VEL
LIN {X 0,Y 632.856,Z 267.388,A -85,B 0,C 180,E1 29117.806,E2 29117.806} C_VEL
LIN {X 0,Y 634.223,Z 270.728,A -85,B 0,C 180,E1 29117.318,E2 29117.318} C_VEL
LIN {X 0,Y 641.584,Z 287.204,A -85,B 0,C 180,E1 29115.153,E2 29115.153} C_VEL
LIN {X 0,Y 654.469,Z 307.247,A -85,B 0,C 180,E1 29113.711,E2 29113.711} C_VEL
LIN {X 0,Y 660.1,Z 316.464,A -85,B 0,C 180,E1 29113.112,E2 29113.112} C_VEL
LIN {X 0,Y 660.824,Z 320.431,A -85,B 0,C 180,E1 29112.995,E2 29112.995} C_VEL
LIN {X 0,Y 656.848,Z 563.089,A -85,B 0,C 180,E1 29109.848,E2 29109.848} C_VEL
LIN {X 0,Y 654.302,Z 720.976,A -85,B 0,C 180,E1 29107.823,E2 29107.823} C_VEL
LIN {X 0,Y 653.359,Z 747.922,A -85,B 0,C 180,E1 29107.33,E2 29107.33} C_VEL
LIN {X 0,Y 652.259,Z 770.204,A -85,B 0,C 180,E1 29106.778,E2 29106.778} C_VEL
LIN {X 0,Y 651.147,Z 789.698,A -85,B 0,C 180,E1 29106.187,E2 29106.187} C_VEL
LIN {X 0,Y 649.835,Z 810.081,A -85,B 0,C 180,E1 29105.456,E2 29105.456} C_VEL
LIN {X 0,Y 648.028,Z 835.187,A -85,B 0,C 180,E1 29104.383,E2 29104.383} C_VEL
LIN {X 0,Y 646.316,Z 856.386,A -85,B 0,C 180,E1 29103.312,E2 29103.312} C_VEL
LIN {X 0,Y 644.581,Z 877.128,A -85,B 0,C 180,E1 29102.116,E2 29102.116} C_VEL
LIN {X 0,Y 642.604,Z 900.062,A -85,B 0,C 180,E1 29100.584,E2 29100.584} C_VEL
LIN {X 0,Y 641.015,Z 917.99,A -85,B 0,C 180,E1 29099.224,E2 29099.224} C_VEL
LIN {X 0,Y 639.326,Z 937.402,A -85,B 0,C 180,E1 29097.577,E2 29097.577} C_VEL
LIN {X 0,Y 637.715,Z 956.238,A -85,B 0,C 180,E1 29095.742,E2 29095.742} C_VEL
LIN {X 0,Y 636.414,Z 972.095,A -85,B 0,C 180,E1 29094.012,E2 29094.012} C_VEL
LIN {X 0,Y 635.096,Z 989.8,A -85,B 0,C 180,E1 29091.812,E2 29091.812} C_VEL
LIN {X 0,Y 634.211,Z 1002.56,A -85,B 0,C 180,E1 29090.006,E2 29090.006} C_VEL
LIN {X 0,Y 633.418,Z 1016.146,A -85,B 0,C 180,E1 29087.833,E2 29087.833} C_VEL
LIN {X 0,Y 632.831,Z 1027.649,A -85,B 0,C 180,E1 29085.675,E2 29085.675} C_VEL
LIN {X 0,Y 632.474,Z 1036.695,A -85,B 0,C 180,E1 29083.718,E2 29083.718} C_VEL
LIN {X 0,Y 632.173,Z 1046.053,A -85,B 0,C 180,E1 29081.311,E2 29081.311} C_VEL
LIN {X 0,Y 632.03,Z 1052.681,A -85,B 0,C 180,E1 29079.18,E2 29079.18} C_VEL
LIN {X 0,Y 631.962,Z 1057.538,A -85,B 0,C 180,E1 29077.232,E2 29077.232} C_VEL
LIN {X 0,Y 631.911,Z 1061.881,A -85,B 0,C 180,E1 29074.902,E2 29074.902} C_VEL
LIN {X 0,Y 631.913,Z 1064.303,A -85,B 0,C 180,E1 29072.721,E2 29072.721} C_VEL
LIN {X 0,Y 631.903,Z 1065.305,A -85,B 0,C 180,E1 29070.816,E2 29070.816} C_VEL
LIN {X 0,Y 631.915,Z 1065.237,A -85,B 0,C 180,E1 29068.912,E2 29068.912} C_VEL
LIN {X 0,Y 631.906,Z 1063.693,A -85,B 0,C 180,E1 29066.553,E2 29066.553} C_VEL
LIN {X 0,Y 631.909,Z 1060.645,A -85,B 0,C 180,E1 29064.37,E2 29064.37} C_VEL
LIN {X 0,Y 631.964,Z 1057.034,A -85,B 0,C 180,E1 29062.546,E2 29062.546} C_VEL
LIN {X 0,Y 632.038,Z 1052.131,A -85,B 0,C 180,E1 29060.622,E2 29060.622} C_VEL
LIN {X 0,Y 632.227,Z 1044.426,A -85,B 0,C 180,E1 29058.228,E2 29058.228} C_VEL
LIN {X 0,Y 632.497,Z 1035.838,A -85,B 0,C 180,E1 29056.085,E2 29056.085} C_VEL
LIN {X 0,Y 632.884,Z 1026.727,A -85,B 0,C 180,E1 29054.138,E2 29054.138} C_VEL
LIN {X 0,Y 633.542,Z 1013.894,A -85,B 0,C 180,E1 29051.791,E2 29051.791} C_VEL
LIN {X 0,Y 634.297,Z 1001.293,A -85,B 0,C 180,E1 29049.805,E2 29049.805} C_VEL
LIN {X 0,Y 635.35,Z 986.253,A -85,B 0,C 180,E1 29047.711,E2 29047.711} C_VEL
LIN {X 0,Y 636.626,Z 969.56,A -85,B 0,C 180,E1 29045.701,E2 29045.701} C_VEL
LIN {X 0,Y 638.024,Z 952.526,A -85,B 0,C 180,E1 29043.872,E2 29043.872} C_VEL
LIN {X 0,Y 639.696,Z 932.974,A -85,B 0,C 180,E1 29042.036,E2 29042.036} C_VEL
LIN {X 0,Y 641.234,Z 915.555,A -85,B 0,C 180,E1 29040.582,E2 29040.582} C_VEL
LIN {X 0,Y 643.14,Z 893.891,A -85,B 0,C 180,E1 29038.977,E2 29038.977} C_VEL
LIN {X 0,Y 644.895,Z 873.425,A -85,B 0,C 180,E1 29037.662,E2 29037.662} C_VEL
LIN {X 0,Y 646.556,Z 853.688,A -85,B 0,C 180,E1 29036.543,E2 29036.543} C_VEL
LIN {X 0,Y 648.505,Z 828.798,A -85,B 0,C 180,E1 29035.324,E2 29035.324} C_VEL
LIN {X 0,Y 649.992,Z 807.515,A -85,B 0,C 180,E1 29034.446,E2 29034.446} C_VEL
LIN {X 0,Y 651.283,Z 787.3,A -85,B 0,C 180,E1 29033.733,E2 29033.733} C_VEL
LIN {X 0,Y 652.665,Z 762.523,A -85,B 0,C 180,E1 29033.009,E2 29033.009} C_VEL
LIN {X 0,Y 653.724,Z 737.556,A -85,B 0,C 180,E1 29032.46,E2 29032.46} C_VEL
LIN {X 0,Y 654.451,Z 715.274,A -85,B 0,C 180,E1 29032.095,E2 29032.095} C_VEL
LIN {X 0,Y 658.227,Z 476.42,A -85,B 0,C 180,E1 29029.038,E2 29029.038} C_VEL
LIN {X 0,Y 660.715,Z 319.012,A -85,B 0,C 180,E1 29026.975,E2 29026.975} C_VEL
LIN {X 0,Y 659.524,Z 315.183,A -85,B 0,C 180,E1 29026.823,E2 29026.823} C_VEL
LIN {X 0,Y 644.464,Z 291.823,A -85,B 0,C 180,E1 29025.204,E2 29025.204} C_VEL
LIN {X 0,Y 641.316,Z 286.673,A -85,B 0,C 180,E1 29024.807,E2 29024.807} C_VEL
LIN {X 0,Y 633.895,Z 270.174,A -85,B 0,C 180,E1 29022.688,E2 29022.688} C_VEL
LIN {X 0,Y 632.847,Z 267.303,A -85,B 0,C 180,E1 29022.281,E2 29022.281} C_VEL
LIN {X 0,Y 632.837,Z 267.125,A -85,B 0,C 180,E1 29019.55,E2 29019.55} C_VEL
LIN {X 0,Y 632.834,Z 267.153,A -85,B 0,C 180,E1 29016.312,E2 29016.312} C_VEL
LIN {X 0,Y 632.827,Z 267.116,A -85,B 0,C 180,E1 29013.574,E2 29013.574} C_VEL
LIN {X 0,Y 632.845,Z 267.139,A -85,B 0,C 180,E1 29010.371,E2 29010.371} C_VEL
LIN {X 0,Y 632.824,Z 267.128,A -85,B 0,C 180,E1 29007.576,E2 29007.576} C_VEL
LIN {X 0,Y 632.866,Z 267.139,A -85,B 0,C 180,E1 29004.453,E2 29004.453} C_VEL
LIN {X 0,Y 632.819,Z 267.149,A -85,B 0,C 180,E1 29001.602,E2 29001.602} C_VEL
LIN {X 0,Y 632.89,Z 267.147,A -85,B 0,C 180,E1 28998.573,E2 28998.573} C_VEL
LIN {X 0,Y 632.818,Z 267.147,A -85,B 0,C 180,E1 28995.582,E2 28995.582} C_VEL
LIN {X 0,Y 632.892,Z 267.134,A -85,B 0,C 180,E1 28992.593,E2 28992.593} C_VEL
LIN {X 0,Y 632.818,Z 267.146,A -85,B 0,C 180,E1 28989.55,E2 28989.55} C_VEL
LIN {X 0,Y 632.887,Z 267.143,A -85,B 0,C 180,E1 28986.623,E2 28986.623} C_VEL
LIN {X 0,Y 632.819,Z 267.145,A -85,B 0,C 180,E1 28983.533,E2 28983.533} C_VEL
LIN {X 0,Y 632.869,Z 267.142,A -85,B 0,C 180,E1 28980.634,E2 28980.634} C_VEL
LIN {X 0,Y 632.824,Z 267.15,A -85,B 0,C 180,E1 28977.555,E2 28977.555} C_VEL
LIN {X 0,Y 632.844,Z 267.138,A -85,B 0,C 180,E1 28974.742,E2 28974.742} C_VEL
LIN {X 0,Y 632.827,Z 267.137,A -85,B 0,C 180,E1 28971.55,E2 28971.55} C_VEL
LIN {X 0,Y 632.832,Z 267.148,A -85,B 0,C 180,E1 28968.794,E2 28968.794} C_VEL
LIN {X 0,Y 632.837,Z 267.152,A -85,B 0,C 180,E1 28965.544,E2 28965.544} C_VEL
LIN {X 0,Y 632.823,Z 267.135,A -85,B 0,C 180,E1 28962.814,E2 28962.814} C_VEL
LIN {X 0,Y 632.856,Z 267.138,A -85,B 0,C 180,E1 28959.66,E2 28959.66} C_VEL
LIN {X 0,Y 632.818,Z 267.149,A -85,B 0,C 180,E1 28956.866,E2 28956.866} C_VEL
LIN {X 0,Y 632.881,Z 267.095,A -85,B 0,C 180,E1 28953.815,E2 28953.815} C_VEL
LIN {X 0,Y 632.817,Z 267.15,A -85,B 0,C 180,E1 28950.879,E2 28950.879} C_VEL
LIN {X 0,Y 632.872,Z 267.112,A -85,B 0,C 180,E1 28948.039,E2 28948.039} C_VEL
LIN {X 0,Y 632.82,Z 267.142,A -85,B 0,C 180,E1 28944.931,E2 28944.931} C_VEL
LIN {X 0,Y 632.856,Z 267.133,A -85,B 0,C 180,E1 28942.076,E2 28942.076} C_VEL
LIN {X 0,Y 632.827,Z 267.137,A -85,B 0,C 180,E1 28939.026,E2 28939.026} C_VEL
LIN {X 0,Y 632.824,Z 267.14,A -85,B 0,C 180,E1 28936.332,E2 28936.332} C_VEL
LIN {X 0,Y 632.894,Z 267.369,A -85,B 0,C 180,E1 28933.91,E2 28933.91} C_VEL
LIN {X 0,Y 636.944,Z 277.132,A -85,B 0,C 180,E1 28932.608,E2 28932.608} C_VEL
LIN {X 0,Y 638.138,Z 280.348,A -85,B 0,C 180,E1 28932.357,E2 28932.357} C_VEL
LIN {X 0,Y 639.563,Z 287.293,A -85,B 0,C 180,E1 28932.115,E2 28932.115} C_VEL
LIN {X 0,Y 641.09,Z 295.165,A -85,B 0,C 180,E1 28931.862,E2 28931.862} C_VEL
LIN {X 0,Y 642.492,Z 298.119,A -85,B 0,C 180,E1 28931.691,E2 28931.691} C_VEL
LIN {X 0,Y 654.877,Z 317.665,A -85,B 0,C 180,E1 28930.34,E2 28930.34} C_VEL
LIN {X 0,Y 650.687,Z 555.228,A -85,B 0,C 180,E1 28927.23,E2 28927.23} C_VEL
LIN {X 0,Y 647.982,Z 711.06,A -85,B 0,C 180,E1 28925.212,E2 28925.212} C_VEL
LIN {X 0,Y 646.974,Z 737.946,A -85,B 0,C 180,E1 28924.718,E2 28924.718} C_VEL
LIN {X 0,Y 645.806,Z 760.201,A -85,B 0,C 180,E1 28924.162,E2 28924.162} C_VEL
LIN {X 0,Y 644.583,Z 780.256,A -85,B 0,C 180,E1 28923.549,E2 28923.549} C_VEL
LIN {X 0,Y 643.057,Z 802.652,A -85,B 0,C 180,E1 28922.732,E2 28922.732} C_VEL
LIN {X 0,Y 641.119,Z 827.164,A -85,B 0,C 180,E1 28921.655,E2 28921.655} C_VEL
LIN {X 0,Y 639.437,Z 846.807,A -85,B 0,C 180,E1 28920.648,E2 28920.648} C_VEL
LIN {X 0,Y 637.59,Z 867.389,A -85,B 0,C 180,E1 28919.448,E2 28919.448} C_VEL
LIN {X 0,Y 635.47,Z 890.169,A -85,B 0,C 180,E1 28917.911,E2 28917.911} C_VEL
LIN {X 0,Y 633.755,Z 908.318,A -85,B 0,C 180,E1 28916.519,E2 28916.519} C_VEL
LIN {X 0,Y 631.926,Z 927.854,A -85,B 0,C 180,E1 28914.841,E2 28914.841} C_VEL
LIN {X 0,Y 630.231,Z 946.06,A -85,B 0,C 180,E1 28913.044,E2 28913.044} C_VEL
LIN {X 0,Y 628.887,Z 961.422,A -85,B 0,C 180,E1 28911.352,E2 28911.352} C_VEL
LIN {X 0,Y 627.451,Z 978.955,A -85,B 0,C 180,E1 28909.164,E2 28909.164} C_VEL
LIN {X 0,Y 626.454,Z 992.232,A -85,B 0,C 180,E1 28907.27,E2 28907.27} C_VEL
LIN {X 0,Y 625.597,Z 1005.692,A -85,B 0,C 180,E1 28905.101,E2 28905.101} C_VEL
LIN {X 0,Y 624.936,Z 1017.573,A -85,B 0,C 180,E1 28902.85,E2 28902.85} C_VEL
LIN {X 0,Y 624.529,Z 1026.527,A -85,B 0,C 180,E1 28900.89,E2 28900.89} C_VEL
LIN {X 0,Y 624.229,Z 1035.546,A -85,B 0,C 180,E1 28898.567,E2 28898.567} C_VEL
LIN {X 0,Y 624.043,Z 1042.424,A -85,B 0,C 180,E1 28896.347,E2 28896.347} C_VEL
LIN {X 0,Y 623.965,Z 1047.244,A -85,B 0,C 180,E1 28894.411,E2 28894.411} C_VEL
LIN {X 0,Y 623.913,Z 1051.11,A -85,B 0,C 180,E1 28892.388,E2 28892.388} C_VEL
LIN {X 0,Y 623.928,Z 1054.156,A -85,B 0,C 180,E1 28889.908,E2 28889.908} C_VEL
LIN {X 0,Y 623.906,Z 1055.279,A -85,B 0,C 180,E1 28887.888,E2 28887.888} C_VEL
LIN {X 0,Y 623.909,Z 1055.263,A -85,B 0,C 180,E1 28885.956,E2 28885.956} C_VEL
LIN {X 0,Y 623.911,Z 1053.897,A -85,B 0,C 180,E1 28883.651,E2 28883.651} C_VEL
LIN {X 0,Y 623.91,Z 1050.789,A -85,B 0,C 180,E1 28881.336,E2 28881.336} C_VEL
LIN {X 0,Y 623.97,Z 1046.981,A -85,B 0,C 180,E1 28879.381,E2 28879.381} C_VEL
LIN {X 0,Y 624.045,Z 1042.016,A -85,B 0,C 180,E1 28877.414,E2 28877.414} C_VEL
LIN {X 0,Y 624.258,Z 1034.164,A -85,B 0,C 180,E1 28874.961,E2 28874.961} C_VEL
LIN {X 0,Y 624.55,Z 1025.871,A -85,B 0,C 180,E1 28872.868,E2 28872.868} C_VEL
LIN {X 0,Y 624.99,Z 1016.565,A -85,B 0,C 180,E1 28870.855,E2 28870.855} C_VEL
LIN {X 0,Y 625.719,Z 1003.452,A -85,B 0,C 180,E1 28868.436,E2 28868.436} C_VEL
LIN {X 0,Y 626.533,Z 991.209,A -85,B 0,C 180,E1 28866.486,E2 28866.486} C_VEL
LIN {X 0,Y 627.657,Z 976.258,A -85,B 0,C 180,E1 28864.379,E2 28864.379} C_VEL
LIN {X 0,Y 628.972,Z 960.433,A -85,B 0,C 180,E1 28862.445,E2 28862.445} C_VEL
LIN {X 0,Y 630.331,Z 944.93,A -85,B 0,C 180,E1 28860.747,E2 28860.747} C_VEL
LIN {X 0,Y 632.245,Z 924.281,A -85,B 0,C 180,E1 28858.753,E2 28858.753} C_VEL
LIN {X 0,Y 633.864,Z 907.161,A -85,B 0,C 180,E1 28857.298,E2 28857.298} C_VEL
LIN {X 0,Y 635.682,Z 887.987,A -85,B 0,C 180,E1 28855.838,E2 28855.838} C_VEL
LIN {X 0,Y 637.797,Z 865.131,A -85,B 0,C 180,E1 28854.325,E2 28854.325} C_VEL
LIN {X 0,Y 639.518,Z 845.934,A -85,B 0,C 180,E1 28853.215,E2 28853.215} C_VEL
LIN {X 0,Y 641.402,Z 824.071,A -85,B 0,C 180,E1 28852.106,E2 28852.106} C_VEL
LIN {X 0,Y 643.239,Z 799.831,A -85,B 0,C 180,E1 28851.069,E2 28851.069} C_VEL
LIN {X 0,Y 644.627,Z 779.529,A -85,B 0,C 180,E1 28850.336,E2 28850.336} C_VEL
LIN {X 0,Y 645.888,Z 758.726,A -85,B 0,C 180,E1 28849.706,E2 28849.706} C_VEL
LIN {X 0,Y 647.168,Z 733.019,A -85,B 0,C 180,E1 28849.085,E2 28849.085} C_VEL
LIN {X 0,Y 648.039,Z 708.742,A -85,B 0,C 180,E1 28848.664,E2 28848.664} C_VEL
LIN {X 0,Y 651.984,Z 479.838,A -85,B 0,C 180,E1 28845.702,E2 28845.702} C_VEL
LIN {X 0,Y 654.72,Z 317.201,A -85,B 0,C 180,E1 28843.55,E2 28843.55} C_VEL
LIN {X 0,Y 639.87,Z 293.988,A -85,B 0,C 180,E1 28841.901,E2 28841.901} C_VEL
LIN {X 0,Y 629.455,Z 278.761,A -85,B 0,C 180,E1 28840.654,E2 28840.654} C_VEL
LIN {X 0,Y 626.296,Z 271.766,A -85,B 0,C 180,E1 28839.688,E2 28839.688} C_VEL
LIN {X 0,Y 624.903,Z 268.293,A -85,B 0,C 180,E1 28839.141,E2 28839.141} C_VEL
LIN {X 0,Y 624.951,Z 268.133,A -85,B 0,C 180,E1 28836.184,E2 28836.184} C_VEL
LIN {X 0,Y 624.878,Z 268.134,A -85,B 0,C 180,E1 28833.179,E2 28833.179} C_VEL
LIN {X 0,Y 624.961,Z 268.112,A -85,B 0,C 180,E1 28830.158,E2 28830.158} C_VEL
LIN {X 0,Y 624.878,Z 268.124,A -85,B 0,C 180,E1 28827.132,E2 28827.132} C_VEL
LIN {X 0,Y 624.952,Z 268.118,A -85,B 0,C 180,E1 28824.079,E2 28824.079} C_VEL
LIN {X 0,Y 624.879,Z 268.116,A -85,B 0,C 180,E1 28821.102,E2 28821.102} C_VEL
LIN {X 0,Y 624.942,Z 268.12,A -85,B 0,C 180,E1 28818.125,E2 28818.125} C_VEL
LIN {X 0,Y 624.878,Z 268.12,A -85,B 0,C 180,E1 28815.024,E2 28815.024} C_VEL
LIN {X 0,Y 624.925,Z 268.111,A -85,B 0,C 180,E1 28812.149,E2 28812.149} C_VEL
LIN {X 0,Y 624.882,Z 268.13,A -85,B 0,C 180,E1 28809.022,E2 28809.022} C_VEL
LIN {X 0,Y 624.899,Z 268.093,A -85,B 0,C 180,E1 28806.247,E2 28806.247} C_VEL
LIN {X 0,Y 624.889,Z 268.136,A -85,B 0,C 180,E1 28803.027,E2 28803.027} C_VEL
LIN {X 0,Y 624.889,Z 268.095,A -85,B 0,C 180,E1 28800.275,E2 28800.275} C_VEL
LIN {X 0,Y 624.893,Z 268.138,A -85,B 0,C 180,E1 28796.973,E2 28796.973} C_VEL
LIN {X 0,Y 624.887,Z 268.109,A -85,B 0,C 180,E1 28794.214,E2 28794.214} C_VEL
LIN {X 0,Y 624.901,Z 268.127,A -85,B 0,C 180,E1 28790.978,E2 28790.978} C_VEL
LIN {X 0,Y 624.887,Z 268.129,A -85,B 0,C 180,E1 28788.181,E2 28788.181} C_VEL
LIN {X 0,Y 624.909,Z 268.106,A -85,B 0,C 180,E1 28784.977,E2 28784.977} C_VEL
LIN {X 0,Y 624.884,Z 268.138,A -85,B 0,C 180,E1 28782.188,E2 28782.188} C_VEL
LIN {X 0,Y 624.936,Z 268.096,A -85,B 0,C 180,E1 28779.096,E2 28779.096} C_VEL
LIN {X 0,Y 624.881,Z 268.141,A -85,B 0,C 180,E1 28776.219,E2 28776.219} C_VEL
LIN {X 0,Y 624.956,Z 268.135,A -85,B 0,C 180,E1 28773.18,E2 28773.18} C_VEL
LIN {X 0,Y 624.884,Z 268.141,A -85,B 0,C 180,E1 28770.262,E2 28770.262} C_VEL
LIN {X 0,Y 624.935,Z 268.086,A -85,B 0,C 180,E1 28767.308,E2 28767.308} C_VEL
LIN {X 0,Y 624.886,Z 268.142,A -85,B 0,C 180,E1 28764.219,E2 28764.219} C_VEL
LIN {X 0,Y 624.929,Z 268.09,A -85,B 0,C 180,E1 28761.273,E2 28761.273} C_VEL
LIN {X 0,Y 624.946,Z 268.369,A -85,B 0,C 180,E1 28758.533,E2 28758.533} C_VEL
LIN {X 0,Y 626.327,Z 271.839,A -85,B 0,C 180,E1 28758.017,E2 28758.017} C_VEL
LIN {X 0,Y 630.736,Z 281.611,A -85,B 0,C 180,E1 28756.652,E2 28756.652} C_VEL
LIN {X 0,Y 633.452,Z 287.422,A -85,B 0,C 180,E1 28755.906,E2 28755.906} C_VEL
LIN {X 0,Y 647.921,Z 309.649,A -85,B 0,C 180,E1 28754.23,E2 28754.23} C_VEL
LIN {X 0,Y 654.837,Z 321.098,A -85,B 0,C 180,E1 28753.475,E2 28753.475} C_VEL
LIN {X 0,Y 651.57,Z 511.602,A -85,B 0,C 180,E1 28750.966,E2 28750.966} C_VEL
LIN {X 0,Y 647.978,Z 720.674,A -85,B 0,C 180,E1 28748.262,E2 28748.262} C_VEL
LIN {X 0,Y 646.997,Z 747.369,A -85,B 0,C 180,E1 28747.775,E2 28747.775} C_VEL
LIN {X 0,Y 645.817,Z 769.984,A -85,B 0,C 180,E1 28747.213,E2 28747.213} C_VEL
LIN {X 0,Y 644.617,Z 789.695,A -85,B 0,C 180,E1 28746.613,E2 28746.613} C_VEL
LIN {X 0,Y 643.22,Z 810.078,A -85,B 0,C 180,E1 28745.877,E2 28745.877} C_VEL
